// TIA Portal project "LogicRoof" (V17)

(* hardware
DEVICE "S7-1500/ET200MP station_1"  S7-1500 station
   slot 0: "Rail_0"  Rack  6ES7 590-1***0-0AA0
   slot 1: "MAIN_PLC"  CPU 1517F-3 PN/DP  6ES7 517-3FP00-0AB0  V2.9
      slot 3: "CPU display_1"  6ES7591-1BA00-0AA0
      slot 32768: "PROFINET interface_1"  X1
         slot 32769: "Port_1"  X1 P1
         slot 32770: "Port_2"  X1 P2
      slot 33024: "PROFINET interface_2"  X2
         slot 33025: "Port_1"  X2 P1
      slot 33280: "DP interface_1"  X3
      slot 34817: "Virtual CP interface port_1"  Virtual CP interface port  Virtual CP interface port
   slot 2: "CP 1543-1_1"  CP 1543-1  6GK7 543-1AX00-0XE0  V3.0
DEVICE "Lift1_PLC"  GSD.Device.PN
   slot 0: "Rack"  Rack  V1.0
   slot 1: "Lift1_PLC"  PLC-Lift1  6ES7 288-1ST60-0AA1  V02.07.00
      slot 0: "PLC-Lift1 Virtual submodule"  PLC-Lift1 Virtual submodule
      slot 1: "传送区01"  传送区01
      slot 2: "传送区02"  传送区02
      slot 3: "Interface"  Interface
         slot 1: "Port 1"  Port 1
DEVICE "Stacker_PLC"  GSD.Device.PN
   slot 0: "Rack"  Rack  V1.0
   slot 1: "Stacker_PLC"  PLC-Stacker  6ES7 288-1ST60-0AA0  V02.05.00
      slot 0: "PLC-Stacker Virtual submodule"  PLC-Stacker Virtual submodule
      slot 1: "传送区01"  传送区01
      slot 2: "传送区02"  传送区02
      slot 3: "Interface"  Interface
         slot 1: "Port 1"  Port 1
DEVICE "MDB_IO"  GSD.Device.PN
   slot 0: "Rack"  Rack  V1.0
   slot 0: "mdb-io"  CN-8032  CN-8032  V1.00
      slot 0: "CN-8032"  CN-8032
      slot 1: "PN-IO"  PN-IO
         slot 1: "Port 1"  Port 1
         slot 2: "Port 2"  Port 2
   slot 1: "DI1"  CT-121F (16DI 24Vdc) Sink Input  CT-121F  V1.00
      slot 0: "16DI Input Status"  16DI Input Status
   slot 1: "16DI Counter Submodule"  16DI Counter Submodule
   slot 1: "16DI Counter Submodule"  16DI Counter Submodule
   slot 2: "DI2"  CT-121F (16DI 24Vdc) Sink Input  CT-121F  V1.00
      slot 0: "16DI Input Status"  16DI Input Status
   slot 3: "DI3"  CT-121F (16DI 24Vdc) Sink Input  CT-121F  V1.00
      slot 0: "16DI Input Status"  16DI Input Status
   slot 4: "DO1"  CT-222F (16DO 24Vdc) Source Output TTL  CT-222F  V1.00
      slot 0: "16DO Output Status"  16DO Output Status
   slot 5: "DO2"  CT-222F (16DO 24Vdc) Source Output TTL  CT-222F  V1.00
      slot 0: "16DO Output Status"  16DO Output Status
DEVICE "SDB_IO"  GSD.Device.PN
   slot 0: "Rack"  Rack  V1.0
   slot 0: "SDB-IO"  CN-8032  CN-8032  V1.00
      slot 0: "CN-8032"  CN-8032
      slot 1: "PN-IO"  PN-IO
         slot 1: "Port 1"  Port 1
         slot 2: "Port 2"  Port 2
   slot 1: "DI1"  CT-121F (16DI 24Vdc) Sink Input  CT-121F  V1.00
      slot 0: "16DI Input Status"  16DI Input Status
   slot 1: "16DI Counter Submodule"  16DI Counter Submodule
   slot 1: "16DI Counter Submodule"  16DI Counter Submodule
   slot 2: "DI2"  CT-121F (16DI 24Vdc) Sink Input  CT-121F  V1.00
      slot 0: "16DI Input Status"  16DI Input Status
   slot 4: "DO1"  CT-222F (16DO 24Vdc) Source Output TTL  CT-222F  V1.00
      slot 0: "16DO Output Status"  16DO Output Status
DEVICE "PU_IO"  GSD.Device.PN
   slot 0: "Rack"  Rack  V1.0
   slot 0: "PU-IO"  CN-8032  CN-8032  V1.00
      slot 0: "CN-8032"  CN-8032
      slot 1: "PN-IO"  PN-IO
         slot 1: "Port 1"  Port 1
         slot 2: "Port 2"  Port 2
   slot 1: "DI1"  CT-121F (16DI 24Vdc) Sink Input  CT-121F  V1.00
      slot 0: "16DI Input Status"  16DI Input Status
   slot 1: "16DI Counter Submodule"  16DI Counter Submodule
   slot 1: "16DI Counter Submodule"  16DI Counter Submodule
   slot 4: "DO1"  CT-222F (16DO 24Vdc) Source Output TTL  CT-222F  V1.00
      slot 0: "16DO Output Status"  16DO Output Status
DEVICE "Lift2_PLC"  GSD.Device.PN
   slot 0: "Rack"  Rack  V1.0
   slot 1: "Lift2_PLC"  PLC-Lift1  6ES7 288-1ST60-0AA1  V02.07.00
      slot 0: "PLC-Lift1 Virtual submodule"  PLC-Lift1 Virtual submodule
      slot 1: "传送区01"  传送区01
      slot 2: "传送区02"  传送区02
      slot 3: "Interface"  Interface
         slot 1: "Port 1"  Port 1
DEVICE "GSD device_1"  GSD.Device.PN
   slot 0: "Rack"  Rack  V1.0
   slot 0: "C8-U1"  ConveyLinx in PLC mode  ERSC  V5.07.00
      slot 0: "ConveyLinx in PLC mode"  ConveyLinx in PLC mode
      slot 1: "Interface"  Interface
         slot 1: "Port 1"  Port 1
         slot 2: "Port 2"  Port 2
      slot 1: "Inputs"  virtual input module 64 byte  NO_ORDER_CODE  1.0
         slot 0: "virtual input module 64 byte"  virtual input module 64 byte
      slot 2: "Outputs"  virtual output module 64 byte  NO_ORDER_CODE  1.0
         slot 0: "virtual output module 64 byte"  virtual output module 64 byte
DEVICE "C1_M1_1"  GSD.Device.PN
   slot 0: "Rack"  Rack  V1.0
   slot 0: "C2-M1"  AD1000PN  AD1000PN
      slot 0: "AD1000PN"  AD1000PN
      slot 1: "Interface"  Interface
         slot 1: "Port 1"  Port 1
         slot 2: "Port 2"  Port 2
   slot 1: "Data"  Standard telegram 3, PZD-6/6
      slot 0: "Standard telegram 3, PZD-6/6"  Standard telegram 3, PZD-6/6
DEVICE "C1_M1_2"  GSD.Device.PN
   slot 0: "Rack"  Rack  V1.0
   slot 0: "C1-M1"  AD1000PN  AD1000PN
      slot 0: "AD1000PN"  AD1000PN
      slot 1: "Interface"  Interface
         slot 1: "Port 1"  Port 1
         slot 2: "Port 2"  Port 2
   slot 1: "Data"  Standard telegram 3, PZD-6/6
      slot 0: "Standard telegram 3, PZD-6/6"  Standard telegram 3, PZD-6/6
*)

// ===== PLC "MAIN_PLC"  CPU 1517F-3 PN/DP =====

VAR_GLOBAL   // PLC tag table "SDB_IO"
   "bSDB_KM1_St" AT %I218.0 : Bool;   // Статус главного контактора
   "bSDB_QF1_St" AT %I218.1 : Bool;   // Статус автоматического выкл. QF1
   "bSDB_QF2_St" AT %I218.2 : Bool;   // Статус автоматического выкл. QF2
   "bSDB_QF3_St" AT %I218.3 : Bool;   // Статус автоматического выкл. QF3
   "bSDB_QF4_St" AT %I218.4 : Bool;   // Статус автоматического выкл. QF4
   "bSDB_QF5_St" AT %I218.5 : Bool;   // Статус автоматического выкл. QF5
   "bSDB_QF6_St" AT %I218.6 : Bool;   // Статус автоматического выкл. QF6
   "bFS_SDB_KSF1_St" AT %I218.7 : Bool;   // Статус реле безопасности KSF1
   "bFS_SDB_SB2_St" AT %I219.0 : Bool;   // Кнопка аварийного останова
   "bFS_SDB_SBR1_St" AT %I219.1 : Bool;   // Кнопка сброса аварии
   "bFS_SR3_St" AT %I219.2 : Bool;   // Трос безопасности SR3
   "bFS_SR3_1_St" AT %I219.3 : Bool;   // Трос безопасности SR3.1
   "bFS_SR3_2_St" AT %I219.4 : Bool;   // Трос безопасности SR3.2
   "bFS_SR3_3_St" AT %I219.5 : Bool;   // Трос безопасности SR3.3
   "bSens_5_D4" AT %I219.6 : Bool;   // Датчик -5-D4
   "bSens_5_D5" AT %I219.7 : Bool;   // Датчик -5-D5
   "bSens_6_D4" AT %I284.0 : Bool;   // Датчик -6-D4
   "bSens_6_D5" AT %I284.1 : Bool;   // Датчик -6-D5
   "bSens_7_D4" AT %I284.2 : Bool;   // Датчик -7-D4
   "bSens_7_D5" AT %I284.3 : Bool;   // Датчик -7-D5
   "bSens_8_D3" AT %I284.4 : Bool;   // Датчик -8-D3
   "bFS_SB4_St" AT %I284.5 : Bool;   // Кнопка аварийного останова SB4
   "bFS_SB5_St" AT %I284.6 : Bool;   // Кнопка аварийного останова SB5
   "bFS_SB6_St" AT %I284.7 : Bool;   // Кнопка аварийного останова SB6
   "bFS_SB7_St" AT %I285.0 : Bool;   // Кнопка аварийного останова SB7
   "bSDB_DI2_9" AT %I285.1 : Bool;   // Резерв
   "bSDB_DI2_10" AT %I285.2 : Bool;   // Резерв
   "bSDB_DI2_11" AT %I285.3 : Bool;   // Резерв
   "bSDB_DI2_12" AT %I285.4 : Bool;   // Резерв
   "bSDB_DI2_13" AT %I285.5 : Bool;   // Резерв
   "bSDB_DI2_14" AT %I285.6 : Bool;   // Резерв
   "bSDB_DI2_15" AT %I285.7 : Bool;   // Резерв
   "bSDB_KM1_Ctrl" AT %Q90.0 : Bool;   // Вкл. главного контактора
   "bFS_SDB_KSF1_Reset" AT %Q90.1 : Bool;   // Сброс реле безопасности (старт)
   "bFS_SDB_SafetyMuting" AT %Q90.2 : Bool;   // Safety muting
   "bFS_Lift1Safety_Reset" AT %Q90.3 : Bool;   // Сброс реле безопасности (старт) Лифта 1
   "bSDB_DO1_4" AT %Q90.4 : Bool;   // Резерв
   "bSDB_DO1_5" AT %Q90.5 : Bool;   // Резерв
   "bSDB_DO1_6" AT %Q90.6 : Bool;   // Резерв
   "bSDB_DO1_7" AT %Q90.7 : Bool;   // Резерв
   "bSDB_GeneralAlarm_Ind" AT %Q91.0 : Bool;   // Общая авария
   "bFS_SDB_SafetyAlarm_Ind" AT %Q91.1 : Bool;   // Авария системы безопасности
   "bFS_SDB_SBR1_HL" AT %Q91.2 : Bool;   // Подсветка кнопки СБРОС
   "bSDB_Light_Red" AT %Q91.3 : Bool;   // Свет. колонна, Красный
   "bSDB_Light_Yellow" AT %Q91.4 : Bool;   // Свет. колонна, Желтый
   "bSDB_Light_Green" AT %Q91.5 : Bool;   // Свет. колонна, Зеленый
   "bSDB_Light_Blue" AT %Q91.6 : Bool;   // Свет. колонна, Синий
   "bSDB_Light_Siren" AT %Q91.7 : Bool;   // Свет. колонна, Сирена
END_VAR

VAR_GLOBAL   // PLC tag table "MDB_IO"
   "bStation1_Pwr_St" AT %I64.0 : Bool;   // Цепь питания станции вызревания 1
   "bStation2_Pwr_St" AT %I64.1 : Bool;   // Цепь питания станции вызревания 2
   "bStation3_Pwr_St" AT %I64.2 : Bool;   // Цепь питания станции вызревания 3
   "bStation4_Pwr_St" AT %I64.3 : Bool;   // Цепь питания станции вызревания 4
   "bStation5_Pwr_St" AT %I64.4 : Bool;   // Цепь питания станции вызревания 5
   "bStation6_Pwr_St" AT %I64.5 : Bool;   // Цепь питания станции вызревания 6
   "bStation7_Pwr_St" AT %I64.6 : Bool;   // Цепь питания станции вызревания 7
   "bStation8_Pwr_St" AT %I64.7 : Bool;   // Цепь питания станции вызревания 8
   "bStation9_Pwr_St" AT %I65.0 : Bool;   // Цепь питания станции вызревания 9
   "bStation10_Pwr_St" AT %I65.1 : Bool;   // Цепь питания станции вызревания 10
   "bStation11_Pwr_St" AT %I65.2 : Bool;   // Цепь питания станции вызревания 11
   "bStation12_Pwr_St" AT %I65.3 : Bool;   // Цепь питания станции вызревания 12
   "bStation13_Pwr_St" AT %I65.4 : Bool;   // Цепь питания станции вызревания 13
   "bStation14_Pwr_St" AT %I65.5 : Bool;   // Цепь питания станции вызревания 14
   "bConv35_36_Pwr_St" AT %I65.6 : Bool;   // Автомат QF15 питания шкафа SDB включен
   "bMDB_QF16_St" AT %I65.7 : Bool;   // Автомат QF16 питания паллетайзера включен
   "bMDB_QF17_St" AT %I150.0 : Bool;   // Автомат QF17 питания лифта 2
   "bMDB_QF18_St" AT %I150.1 : Bool;   // Автомат QF18 питания секций 35, 36
   "bMDB_K1_St" AT %I150.2 : Bool;   // Реле контроля фаз K1
   "bFS_MDB_KSF1_St" AT %I150.3 : Bool;   // Статус реле безопасности KSF1
   "bFS_MDB_KSF2_St" AT %I150.4 : Bool;   // Статус реле безопасности KSF2
   "bFS_MDB_KSF3_St" AT %I150.5 : Bool;   // Статус реле безопасности KSF3
   "bFS_MDB_SB1_St" AT %I150.6 : Bool;   // Кнопка аварийного останова SB1
   "bFS_MDB_SBR1_St" AT %I150.7 : Bool;   // Кнопка сброса аварии SBR1
   "bFS_SR1_St" AT %I151.0 : Bool;   // Трос безопасности SR1
   "bFS_SR1_1_St" AT %I151.1 : Bool;   // Трос безопасности SR1.1
   "bFS_SR1_2_St" AT %I151.2 : Bool;   // Трос безопасности SR1.2
   "bFS_SR1_3_St" AT %I151.3 : Bool;   // Трос безопасности SR1.3
   "bFS_SR2_St" AT %I151.4 : Bool;   // Трос безопасности SR2
   "bFS_SR2_1_St" AT %I151.5 : Bool;   // Трос безопасности SR2.1
   "bFS_SR2_2_St" AT %I151.6 : Bool;   // Трос безопасности SR2.2
   "bFS_SR2_3_St" AT %I151.7 : Bool;   // Трос безопасности SR2.3
   "bSens_37_D1" AT %I216.0 : Bool;   // Датчик 37-D1
   "bSens_37_D2" AT %I216.1 : Bool;   // Датчик 37-D2
   "bSens_37_D4" AT %I216.2 : Bool;   // Датчик 37-D4
   "bSens_37_D5" AT %I216.3 : Bool;   // Датчик 37-D5
   "bSens_37_D3" AT %I216.4 : Bool;   // Датчик 37-D3
   "bMDB_DI3_5" AT %I216.5 : Bool;   // Резерв 1
   "bMDB_DI3_6" AT %I216.6 : Bool;   // Резерв 2
   "bMDB_DI3_7" AT %I216.7 : Bool;   // Резерв 3
   "bMDB_DI3_8" AT %I217.0 : Bool;   // Резерв 4
   "bMDB_DI3_9" AT %I217.1 : Bool;   // Резерв 5
   "bMDB_DI3_10" AT %I217.2 : Bool;   // Резерв 6
   "bMDB_DI3_11" AT %I217.3 : Bool;   // Резерв 7
   "bMDB_DI3_12" AT %I217.4 : Bool;   // Резерв 8
   "bMDB_DI3_13" AT %I217.5 : Bool;   // Резерв 9
   "bMDB_DI3_14" AT %I217.6 : Bool;   // Резерв 10
   "bMDB_DI3_15" AT %I217.7 : Bool;   // Резерв 11
   "bStation1_Pwr_Ctrl" AT %Q82.0 : Bool;   // Вкл. cтанции вызревания 1
   "bStation2_Pwr_Ctrl" AT %Q82.1 : Bool;   // Вкл. cтанции вызревания 2
   "bStation3_Pwr_Ctrl" AT %Q82.2 : Bool;   // Вкл. cтанции вызревания 3
   "bStation4_Pwr_Ctrl" AT %Q82.3 : Bool;   // Вкл. cтанции вызревания 4
   "bStation5_Pwr_Ctrl" AT %Q82.4 : Bool;   // Вкл. cтанции вызревания 5
   "bStation6_Pwr_Ctrl" AT %Q82.5 : Bool;   // Вкл. cтанции вызревания 6
   "bStation7_Pwr_Ctrl" AT %Q82.6 : Bool;   // Вкл. cтанции вызревания 7
   "bStation8_Pwr_Ctrl" AT %Q82.7 : Bool;   // Вкл. cтанции вызревания 8
   "bStation9_Pwr_Ctrl" AT %Q83.0 : Bool;   // Вкл. cтанции вызревания 9
   "bStation10_Pwr_Ctrl" AT %Q83.1 : Bool;   // Вкл. cтанции вызревания 10
   "bStation11_Pwr_Ctrl" AT %Q83.2 : Bool;   // Вкл. cтанции вызревания 11
   "bStation12_Pwr_Ctrl" AT %Q83.3 : Bool;   // Вкл. cтанции вызревания 12
   "bStation13_Pwr_Ctrl" AT %Q83.4 : Bool;   // Вкл. cтанции вызревания 13
   "bStation14_Pwr_Ctrl" AT %Q83.5 : Bool;   // Вкл. cтанции вызревания 14
   "bConv35_36_Pwr_Ctrl" AT %Q83.6 : Bool;   // Вкл. трансфера и ролик.конвейера
   "bMDB_DO1_15" AT %Q83.7 : Bool;   // Резерв
   "bMDB_GeneralAlarm_Ind" AT %Q84.0 : Bool;   // Общая авария
   "bFS_MDB_SafetyAlarm_Ind" AT %Q84.1 : Bool;   // Авария системы безопасности
   "bFS_MDB_SBR1_HL" AT %Q84.2 : Bool;   // Подсветка кнопки "Сброс"
   "bMDB_Light_Red" AT %Q84.3 : Bool;   // Свет. колонна, Красный
   "bMDB_Light_Yellow" AT %Q84.4 : Bool;   // Свет. колонна, Желтый
   "bMDB_Light_Green" AT %Q84.5 : Bool;   // Свет. колонна, Зеленый
   "bMDB_Light_Blue" AT %Q84.6 : Bool;   // Свет. колонна, Синий
   "bMDB_Light_Siren" AT %Q84.7 : Bool;   // Свет. колонна, Сирена
   "bFS_MDB_KSF1_2_Reset" AT %Q85.0 : Bool;   // Сброс реле безопасности (старт) KSF1 и KSF2
   "bFS_MDB_KSF3_Reset" AT %Q85.1 : Bool;   // Сброс реле безопасности (старт) KSF3
   "bFS_MDB_SafetyMuting" AT %Q85.2 : Bool;   // Safety muting
   "bFS_Lift2Safety_Reset" AT %Q85.3 : Bool;   // Сброс реле безопасности (старт) Лифта 2
   "bFS_StackerSafety_Reset" AT %Q85.4 : Bool;   // Сброс реле безопасности (старт) трехкоординатного стекера
   "bMDB_DO2_13" AT %Q85.5 : Bool;   // Резерв
   "bMDB_DO2_14" AT %Q85.6 : Bool;   // Резерв
   "bMDB_DO2_15" AT %Q85.7 : Bool;   // Резерв
END_VAR

VAR_GLOBAL   // PLC tag table "PU_IO"
   "bFS_PU_SB3_St" AT %I4.0 : Bool;   // Кнопка аварийного останова
   "bFS_PU_SBR1_St" AT %I4.1 : Bool;   // Кнопка сброса аварии
   "bSens_3_S1" AT %I4.2 : Bool;   // Датчик -3-S1
   "bSens_3_S2" AT %I4.3 : Bool;   // Датчик -3-S2
   "bPU_DI1_4" AT %I4.4 : Bool;   // Резерв
   "bPU_DI1_5" AT %I4.5 : Bool;   // Резерв
   "bPU_DI1_6" AT %I4.6 : Bool;   // Резерв
   "bPU_DI1_7" AT %I4.7 : Bool;   // Резерв
   "bPU_DI1_8" AT %I5.0 : Bool;   // Резерв
   "bPU_DI1_9" AT %I5.1 : Bool;   // Резерв
   "bPU_DI1_10" AT %I5.2 : Bool;   // Резерв
   "bPU_DI1_11" AT %I5.3 : Bool;   // Резерв
   "bPU_DI1_12" AT %I5.4 : Bool;   // Резерв
   "bPU_DI1_13" AT %I5.5 : Bool;   // Резерв
   "bPU_DI1_14" AT %I5.6 : Bool;   // Резерв
   "bPU_DI1_15" AT %I5.7 : Bool;   // Резерв
   "bPU_GeneralAlarm_Ind" AT %I6.0 : Bool;   // Общая авария
   "bFS_PU_SafetyAlarm_Ind" AT %I6.1 : Bool;   // Авария системы безопасности
   "bFS_PU_SBR1_HL" AT %I6.2 : Bool;   // Подсветка кнопки СБРОС
   "bPU_DO1_3" AT %I6.3 : Bool;   // Резерв
   "bPU_DO1_4" AT %I6.4 : Bool;   // Резерв
   "bPU_DO1_5" AT %I6.5 : Bool;   // Резерв
   "bPU_DO1_6" AT %I6.6 : Bool;   // Резерв
   "bPU_DO1_7" AT %I6.7 : Bool;   // Резерв
   "bPU_DO1_8" AT %I7.0 : Bool;   // Резерв
   "bPU_DO1_9" AT %I7.1 : Bool;   // Резерв
   "bPU_DO1_10" AT %I7.2 : Bool;   // Резерв
   "bPU_DO1_11" AT %I7.3 : Bool;   // Резерв
   "bPU_DO1_12" AT %I7.4 : Bool;   // Резерв
   "bPU_DO1_13" AT %I7.5 : Bool;   // Резерв
   "bPU_DO1_14" AT %I7.6 : Bool;   // Резерв
   "bPU_DO1_15" AT %I7.7 : Bool;   // Резерв
END_VAR

VAR_GLOBAL   // PLC tag table "Drives"
   "Drive01_M1" AT %I0.0 : "stDriveType";
END_VAR

VAR_GLOBAL   // PLC tag table "Global"
   "bResetAlarm" AT %M0.0 : Bool;
   "bRd" AT %M0.1 : Bool;
   "vrRec" AT %MW12 : Word;
   "Tag_1" AT %MW14 : Int;
   "Tag_2" AT %MW16 : Int;
END_VAR

TYPE "stOutbound"
   STRUCT
      bMove : Bool;
      bAllowMove : Bool;
      byConvStatus : Byte;
      bReverse : Bool;
   END_STRUCT;
END_TYPE

TYPE "stDriveType"
   STRUCT
      bDrive : Bool;   // Drive forward output
      bDriveRev : Bool;   // Drive reverse output
      bLowSpeed : Bool;   // Low speed select
      bAlarm : Bool;   // General alarm
      bButtDrive : Bool;   // Manual drive button
      bButtDriveRev : Bool;   // Manual reverse drive button
      bLock : Bool;   // Locking motor
      bSafety : Bool;
      bSwitch : Bool;
      bReadyToRun : Bool;
      bNotReady : Bool;
   END_STRUCT;
END_TYPE

TYPE "stModeType"
   STRUCT
      bAutomat : Bool;   // Auto mode
      bStartAutomat : Bool;   // Auto starting mode
      bStop : Bool;   // Stop mode
      bManual : Bool;   // Manual mode
      bReset : Bool;   // Reset mode
      bResetAlarm : Bool;   // Reset alarms
      bAlarm : Bool;   // Alarm mode
      bReadyToReset : Bool;   // Ready to reset mode
   END_STRUCT;
END_TYPE

TYPE "stDriveIOType"
   STRUCT
      uiIn1 : Int;
      uiIn2 : Int;
      uiIn3 : Int;
      uiIn4 : Int;
      uiIn5 : Int;
      uiIn6 : Int;
      uiOut1 : Int;
      uiOut2 : Int;
      uiOut3 : Int;
      uiOut4 : Int;
      uiOut5 : Int;
      uiOut6 : Int;
   END_STRUCT;
END_TYPE

TYPE "stOutboundRev"
   STRUCT
      bMove : Bool;
      bAllowMove : Bool;
      bMoveRev : Bool;
      bAllowMoveRev : Bool;
      byConvStatus : Byte;
      bReverse : Bool;
   END_STRUCT;
END_TYPE

// folder: FB_DB

DATA_BLOCK "FB_Light_DB"   // DB19
{ S7_Optimized_Access := 'TRUE' }
VERSION : 0.1
// stored: InstanceOfName FB_Light
"FB_Light"
BEGIN
END_DATA_BLOCK

DATA_BLOCK "FB_Mode_DB"   // DB20
{ S7_Optimized_Access := 'TRUE' }
VERSION : 0.1
// stored: InstanceOfName FB_Mode
"FB_Mode"
BEGIN
END_DATA_BLOCK

DATA_BLOCK "FB_SystemTime_DB"   // DB24
{ S7_Optimized_Access := 'TRUE' }
VERSION : 0.1
// stored: InstanceOfName FB_SystemTime
"FB_SystemTime"
BEGIN
END_DATA_BLOCK

// folder: FB_DB/Conv

DATA_BLOCK "fbConv_001"   // DB21
{ S7_Optimized_Access := 'TRUE' }
VERSION : 0.1
// stored: InstanceOfName FB_DirectSection
"FB_DirectSection"
BEGIN
END_DATA_BLOCK

DATA_BLOCK "fbConv_002"   // DB22
{ S7_Optimized_Access := 'TRUE' }
VERSION : 0.1
// stored: InstanceOfName FB_DirectSection
"FB_DirectSection"
BEGIN
END_DATA_BLOCK

DATA_BLOCK "fbConv_010"   // DB23
{ S7_Optimized_Access := 'TRUE' }
VERSION : 0.1
// stored: InstanceOfName FB_DirectSection
"FB_DirectSection"
BEGIN
END_DATA_BLOCK

DATA_BLOCK "fbConv_004"   // DB25
{ S7_Optimized_Access := 'TRUE' }
VERSION : 0.1
// stored: InstanceOfName FB_DirectSectionRev
"FB_DirectSectionRev"
BEGIN
END_DATA_BLOCK

DATA_BLOCK "fbConv_003"   // DB26
{ S7_Optimized_Access := 'TRUE' }
VERSION : 0.1
// stored: InstanceOfName FB_RotarySection
"FB_RotarySection"
BEGIN
END_DATA_BLOCK

DATA_BLOCK "fbConv_009"   // DB27
{ S7_Optimized_Access := 'TRUE' }
VERSION : 0.1
// stored: InstanceOfName FB_DirectSection
"FB_DirectSection"
BEGIN
END_DATA_BLOCK

// folder: Safety

DATA_BLOCK "FB_SafetyGroup_DB"   // DB4
{ S7_Optimized_Access := 'TRUE' }
VERSION : 0.1
// stored: InstanceOfName FB_SafetyGroup
"FB_SafetyGroup"
BEGIN
END_DATA_BLOCK

// folder: Safety/PWR

DATA_BLOCK "FB_Station1Pwr_DB"   // DB1
{ S7_Optimized_Access := 'TRUE' }
VERSION : 0.1
// stored: InstanceOfName FB_PowerGroup
"FB_PowerGroup"
BEGIN
END_DATA_BLOCK

DATA_BLOCK "FB_Station2Pwr_DB"   // DB2
{ S7_Optimized_Access := 'TRUE' }
VERSION : 0.1
// stored: InstanceOfName FB_PowerGroup
"FB_PowerGroup"
BEGIN
END_DATA_BLOCK

DATA_BLOCK "FB_Station7Pwr_DB"   // DB3
{ S7_Optimized_Access := 'TRUE' }
VERSION : 0.1
// stored: InstanceOfName FB_PowerGroup
"FB_PowerGroup"
BEGIN
END_DATA_BLOCK

DATA_BLOCK "FB_Station8Pwr_DB"   // DB5
{ S7_Optimized_Access := 'TRUE' }
VERSION : 0.1
// stored: InstanceOfName FB_PowerGroup
"FB_PowerGroup"
BEGIN
END_DATA_BLOCK

DATA_BLOCK "FB_Station9Pwr_DB"   // DB6
{ S7_Optimized_Access := 'TRUE' }
VERSION : 0.1
// stored: InstanceOfName FB_PowerGroup
"FB_PowerGroup"
BEGIN
END_DATA_BLOCK

DATA_BLOCK "FB_Station10Pwr_DB"   // DB7
{ S7_Optimized_Access := 'TRUE' }
VERSION : 0.1
// stored: InstanceOfName FB_PowerGroup
"FB_PowerGroup"
BEGIN
END_DATA_BLOCK

DATA_BLOCK "FB_Station11Pwr_DB"   // DB8
{ S7_Optimized_Access := 'TRUE' }
VERSION : 0.1
// stored: InstanceOfName FB_PowerGroup
"FB_PowerGroup"
BEGIN
END_DATA_BLOCK

DATA_BLOCK "FB_Station12Pwr_DB"   // DB9
{ S7_Optimized_Access := 'TRUE' }
VERSION : 0.1
// stored: InstanceOfName FB_PowerGroup
"FB_PowerGroup"
BEGIN
END_DATA_BLOCK

DATA_BLOCK "FB_Station13Pwr_DB"   // DB10
{ S7_Optimized_Access := 'TRUE' }
VERSION : 0.1
// stored: InstanceOfName FB_PowerGroup
"FB_PowerGroup"
BEGIN
END_DATA_BLOCK

DATA_BLOCK "FB_Conv35_36Pwr_DB"   // DB11
{ S7_Optimized_Access := 'TRUE' }
VERSION : 0.1
// stored: InstanceOfName FB_PowerGroup
"FB_PowerGroup"
BEGIN
END_DATA_BLOCK

DATA_BLOCK "FB_Station5Pwr_DB"   // DB12
{ S7_Optimized_Access := 'TRUE' }
VERSION : 0.1
// stored: InstanceOfName FB_PowerGroup
"FB_PowerGroup"
BEGIN
END_DATA_BLOCK

DATA_BLOCK "FB_SDB_KM1Pwr_DB"   // DB13
{ S7_Optimized_Access := 'TRUE' }
VERSION : 0.1
// stored: InstanceOfName FB_PowerGroup
"FB_PowerGroup"
BEGIN
END_DATA_BLOCK

DATA_BLOCK "FB_Station3Pwr_DB"   // DB14
{ S7_Optimized_Access := 'TRUE' }
VERSION : 0.1
// stored: InstanceOfName FB_PowerGroup
"FB_PowerGroup"
BEGIN
END_DATA_BLOCK

DATA_BLOCK "FB_Station14Pwr_DB"   // DB15
{ S7_Optimized_Access := 'TRUE' }
VERSION : 0.1
// stored: InstanceOfName FB_PowerGroup
"FB_PowerGroup"
BEGIN
END_DATA_BLOCK

DATA_BLOCK "FB_Station4Pwr_DB"   // DB16
{ S7_Optimized_Access := 'TRUE' }
VERSION : 0.1
// stored: InstanceOfName FB_PowerGroup
"FB_PowerGroup"
BEGIN
END_DATA_BLOCK

DATA_BLOCK "FB_Station6Pwr_DB"   // DB17
{ S7_Optimized_Access := 'TRUE' }
VERSION : 0.1
// stored: InstanceOfName FB_PowerGroup
"FB_PowerGroup"
BEGIN
END_DATA_BLOCK

// folder: System blocks/Program resources

DATA_BLOCK "FB_StartTimer_DB"   // DB18
{ S7_Optimized_Access := 'TRUE' }
AUTHOR : Simatic
FAMILY : IEC
NAME : IEC_TMR
VERSION : 1.0
// stored: InstanceOfName IEC_TIMER
"IEC_TIMER"
BEGIN
END_DATA_BLOCK

// folder: (top level)

FUNCTION_BLOCK "FB_DirectSection_OLD"   // FB13, SCL
{ S7_Optimized_Access := 'FALSE' }
VERSION : 0.1
   VAR_INPUT
      bStartAutomat : Bool;
      bFinalConv : Bool := true;
      bFinalConvReverse : Bool := true;
      bAutomat : Bool;
      bEnable1 : Bool;
      tStartTimer : Time := T#20s;
      bEnable2 : Bool;
      bEnable3 : Bool;
      bEnable4 : Bool;
      ConvStatusPrev : Byte;
      ConvStatusNext : Byte;
      bManual : Bool;
      bDriveAuto : Bool;
      bDriveAutoReverse : Bool;
      bButtManu : Bool;
      bButtManuReverse : Bool;
      bButtMove : Bool;
      bButtMoveReverse : Bool;
      bSens : Bool;
      bSens2 : Bool;
      bSens3 : Bool := true;
      bSensFork : Bool;
      tBusy : Time := T#0.01s;
      tFree : Time := T#3s;
      tLongMove : Time := T#40s;
      bReset : Bool;
      bStop : Bool;
      bReverse : Bool;
      bCurtaineUp : Bool := true;
   END_VAR
   VAR_OUTPUT
      bDrive : Bool;
      bDriveReverse : Bool;
      ConvStatus : Byte;
      bDrivePrev : Bool;
      bLongMoveReverse : Bool;
      bLongMove : Bool;
      bDriveNext : Bool;
      bMovePerm : Bool;
      bMovePermRev : Bool;
   END_VAR
   VAR_IN_OUT
      bMove : Bool;
      bMoveReverse : Bool;
   END_VAR
   VAR
      bDriveManu : Bool;
      bResManu : Bool;
      bDriveManuReverse : Bool;
      bDriveConv : Bool;
      bOnMove : Bool;
      bOffMove : Bool;
      bDriveConvReverse : Bool;
      bOnMoveReverse : Bool;
      bOffMoveReverse : Bool;
      bStartConv : Bool;
      bStartConvReverse : Bool;
      fbBusy1 : "FB_Busy1_LAD";
      fbBusy2 : "FB_Busy1_LAD";
      fbBusy3 : "FB_Busy1_LAD";
      fbBusyFork : "FB_Busy2_LAD";
      fbButt : "FB_Button";
      fbButtReverse : "FB_Button";
      fbLongMove : TON_TIME;
      fbLongMoveReverse : TON_TIME;
      fbButtMove : "FB_r_trig";
      fbButtMoveReverse : "FB_r_trig";
      fbStartAutomat : "FB_r_trig";
      fbConvBusy1Puls : "FB_r_trig";
      fbConvBusy2Puls : "FB_r_trig";
      fbStartTimer : TON_TIME;
      fbStartTimerReverse : TON_TIME;
   END_VAR
BEGIN
   #fbBusy1(bSens:= #bSens,  tFree:=  #tFree ,   tBusy:= #tBusy , Reset := #bReset );
   #fbBusy2(bSens:= #bSens2,  tFree:=   #tFree ,   tBusy:=  #tBusy , Reset := #bReset);
   #fbBusy3( bSens:= #bSens3,  tFree:=   #tFree ,   tBusy:=  #tBusy , Reset := #bReset);
   #fbBusyFork(bSens:= #bSensFork,  tFree:=   T#5s ,   tBusy:= T#0s , Reset := #bReset);

   IF NOT #fbBusy1.ConvBusy AND NOT #fbBusy2.ConvBusy AND #bSens3 THEN
       #ConvStatus := 0;
   ELSIF #fbBusy1.ConvBusy AND NOT #fbBusy2.ConvBusy THEN
       #ConvStatus := 1;
   ELSIF NOT #fbBusy1.ConvBusy AND #fbBusy2.ConvBusy THEN
       #ConvStatus := 2;
   ELSIF #fbBusy1.ConvBusy AND #fbBusy2.ConvBusy THEN
       #ConvStatus := 3;
   END_IF;

   #bDrive := NOT #bStop AND (#bDriveAuto OR #bDriveConv OR #bDriveManu OR #bStartConv);
   #bDriveReverse := NOT #bStop AND (#bDriveAutoReverse OR #bDriveConvReverse OR #bDriveManuReverse OR #bStartConvReverse);

   #bResManu := #bReset OR NOT #bManual;
   #fbButt(bBut:=#bButtManu AND #bManual AND NOT #bDriveManuReverse,
           bRS:= #bResManu,
           bOutB=>#bDriveManu);
   #fbButtReverse(bBut:=#bButtManuReverse AND #bManual  AND NOT #bDriveManu,
                  bRS:=#bResManu,
                  bOutB=>#bDriveManuReverse);
   (*перемещение*)
   (* условия включения перемещения*)
   #bMovePerm := #bAutomat AND #bEnable1 AND #bEnable2 AND (#ConvStatusPrev = 2 OR #ConvStatusPrev = 3) AND #ConvStatus = 0 AND NOT #fbBusyFork.ConvBusy AND NOT #bReverse;
   IF #bMovePerm AND #bCurtaineUp
   THEN
       #bMove := TRUE;
   END_IF;
   (* условия включения обратного перемещения *)
   #bMovePermRev := #bAutomat AND #bEnable3 AND #bEnable4 AND (#ConvStatusNext = 1 OR #ConvStatusNext = 3) AND #ConvStatus = 0 AND NOT #fbBusyFork.ConvBusy AND #bReverse;
   IF #bMovePermRev AND #bCurtaineUp
   THEN
       #bMoveReverse := TRUE;
   END_IF;
   (* включение двигателей *)
   #bDriveConv := NOT #bStop AND #bMove AND NOT (#ConvStatus = 2 OR #ConvStatus = 3);
   #bDrivePrev := NOT #bStop AND #bMove AND NOT (#ConvStatus = 2 OR #ConvStatus = 3) AND NOT (#ConvStatusPrev = 0);
   (* включение двигателей при реверсе*)
   #bDriveConvReverse := NOT #bStop AND #bMoveReverse AND NOT (#ConvStatus = 1 OR #ConvStatus = 3);
   #bDriveNext := NOT #bStop AND #bMoveReverse AND NOT (#ConvStatus = 1 OR #ConvStatus = 3) AND NOT (#ConvStatusNext = 0);
   (* выключение перемещения*)
   IF #bMove AND #ConvStatusPrev = 0 AND (#ConvStatus = 2 OR #ConvStatus = 3) THEN
       #bMove := FALSE;
   END_IF;
   (* выключение перемещения при реверсе*)
   IF #bMoveReverse AND #ConvStatusNext = 0 AND (#ConvStatus = 1 OR #ConvStatus = 3) THEN
       #bMoveReverse := FALSE;
   END_IF;
   (* долгое перемещение*)
   #fbLongMove(IN:=NOT #bStop AND #bMove ,
               PT:=#tLongMove,
               Q=>#bLongMove);
   (* долгое перемещение при реверсе*)
   #fbLongMoveReverse(IN:=NOT #bStop AND #bMoveReverse,
                      PT:=#tLongMove,
                      Q=>#bLongMoveReverse);
   (* включение-выключение перемещения кнопкой*)
   #fbButtMove(CLK:=#bButtMove);
   IF #fbButtMove.Q AND NOT #bMove THEN
       #bOnMove := TRUE;
   END_IF;
   IF #fbButtMove.Q AND #bMove THEN
       #bOffMove := TRUE;
   END_IF;
   IF #bOnMove AND NOT #fbButtMove.Q THEN
       #bMove := TRUE;
       #bOnMove := FALSE;
   END_IF;
   IF #bOffMove AND NOT #fbButtMove.Q THEN
       #bMove := FALSE;
       #bOffMove := FALSE;
   END_IF;
   (* включение-выключение перемещения кнопкой при реверсе*)
   #fbButtMoveReverse(CLK:=#bButtMoveReverse);
   IF #fbButtMoveReverse.Q AND NOT #bMoveReverse THEN
       #bOnMoveReverse := TRUE;
   END_IF;
   IF #fbButtMoveReverse.Q AND #bMoveReverse THEN
       #bOffMoveReverse := TRUE;
   END_IF;
   IF #bOnMoveReverse AND NOT #fbButtMoveReverse.Q THEN
       #bMoveReverse := TRUE;
       #bOnMoveReverse := FALSE;
   END_IF;
   IF #bOffMoveReverse AND NOT #fbButtMoveReverse.Q THEN
       #bMoveReverse := FALSE;
       #bOffMoveReverse := FALSE;
   END_IF;

   IF #bReset THEN
       #bMove := FALSE;
       #bMoveReverse := FALSE;
       #bStartConv := FALSE;
       #bStartConvReverse := FALSE;
   END_IF;

   (* Начальный режим*)
   #fbStartAutomat(CLK:=#bStartAutomat);
   IF #fbStartAutomat.Q AND #bCurtaineUp THEN
       IF NOT #bReverse THEN
           #bStartConv := TRUE;
       ELSE
           #bStartConvReverse := TRUE;
       END_IF;
   END_IF;
   #fbConvBusy1Puls(CLK:=#fbBusy1.ConvBusy);
   #fbConvBusy2Puls(CLK:=#fbBusy2.ConvBusy);
   #fbStartTimer(IN:=#bStartConv,
                 PT:=#tStartTimer);
   #fbStartTimerReverse(IN:=#bStartConvReverse,
                        PT:=#tStartTimer);

   IF (#bFinalConv AND (#ConvStatus = 3 OR #ConvStatus = 2) OR NOT #bFinalConv AND ((#ConvStatus = 3 OR #ConvStatus = 2) AND (#ConvStatusNext = 3 OR #ConvStatusNext = 2)) OR #fbConvBusy2Puls.Q OR #fbStartTimer.Q)
       OR NOT #bStartAutomat
   THEN
       #bStartConv := FALSE;
   END_IF;

   IF (#bStartConvReverse AND (#bFinalConvReverse AND (#ConvStatus = 3 OR #ConvStatus = 1) OR NOT #bFinalConvReverse AND ((#ConvStatus = 3 OR #ConvStatus = 1) AND (#ConvStatusPrev = 3 OR #ConvStatusPrev = 1)) OR #fbConvBusy1Puls.Q OR #fbStartTimerReverse.Q))
       OR NOT #bStartAutomat
   THEN
       #bStartConvReverse := FALSE;
   END_IF;
END_FUNCTION_BLOCK

FUNCTION "FN_IsFree" : Bool   // FC1, SCL
{ S7_Optimized_Access := 'TRUE' }
VERSION : 0.1
   VAR_INPUT
      byConvStatus : Byte;
   END_VAR
BEGIN
   IF #byConvStatus = 0 THEN
       #FN_IsFree := true;
   ELSE
       #FN_IsFree := false;
   END_IF;
   RETURN;
END_FUNCTION

FUNCTION "FN_ConvState" : Byte   // FC2, SCL
{ S7_Optimized_Access := 'TRUE' }
VERSION : 0.1
   VAR_INPUT
      bAuto : Bool;
      bMan : Bool;
      bDrive : Bool;
      bDriveRev : Bool;
      bAlarm : Bool;
   END_VAR
   VAR_TEMP
      byVal : Byte;
   END_VAR
BEGIN
   #byVal := 0;
   IF NOT #bAlarm THEN
       IF #bAuto THEN
           IF #bDrive THEN
               #byVal := 1;
           ELSIF #bDriveRev THEN
               #byVal := 2;
           END_IF;
       ELSE
           IF #bDrive THEN
               #byVal := 3;
           ELSIF #bDriveRev THEN
               #byVal := 4;
           END_IF;
       END_IF;
   ELSE
       #byVal := 5;
   END_IF;
   #FN_ConvState:=#byVal;
   RETURN;
END_FUNCTION

ORGANIZATION_BLOCK "Main"   // OB1, SCL, ProgramCycle
TITLE = "Main Program Sweep (Cycle)"
{ S7_Optimized_Access := 'TRUE' }
VERSION : 0.1
   VAR_INPUT
      Initial_Call : Bool;   // Initial call of this OB
      Remanence : Bool;   // =True, if remanent data are available
   END_VAR
BEGIN
   "FB_SystemTime_DB"();


   "FB_Mode_DB"();
   "FB_Light_DB"(stMode:="FB_Mode_DB".stMode);
   "bMDB_Light_Blue" := "bSDB_Light_Blue" := "FB_Light_DB".bBlue;
   "bMDB_Light_Green" := "bSDB_Light_Green" := "FB_Light_DB".bGreen;
   "bMDB_Light_Yellow" := "bSDB_Light_Yellow" := "FB_Light_DB".bYellow;
   "bMDB_Light_Red" := "bSDB_Light_Red" := "FB_Light_DB".bRed;
   "bMDB_Light_Siren" := "bSDB_Light_Siren" := "FB_Light_DB".bSiren;
END_ORGANIZATION_BLOCK

ORGANIZATION_BLOCK "InboundZone"   // OB123, SCL, ProgramCycle
TITLE = "Main Program Sweep (Cycle)"
{ S7_Optimized_Access := 'TRUE' }
VERSION : 0.1
   VAR_INPUT
      Initial_Call : Bool;   // Initial call of this OB
      Remanence : Bool;   // =True, if remanent data are available
   END_VAR
BEGIN
   "fbConv_001"(wDriveHW_M1:="C1-M1~Data",
                stNext:="fbConv_002".stOut,
                stMode := "FB_Mode_DB".stMode);

   "fbConv_002"(wDriveHW_M1:="C2-M1~Data",
                stNext:="fbConv_003".stOutLine,
                stPrev:="fbConv_001".stOut,
                stMode := "FB_Mode_DB".stMode);

   "fbConv_003"(stNextLine:="fbConv_004".stOut,
                stNextCross:="fbConv_009".stOut,
                stPrevLine:="fbConv_002".stOut,
                stNextLineRev:="fbConv_004".stOutRev,
                stMode:="FB_Mode_DB".stMode);

   "fbConv_004"(stPrev := "fbConv_003".stOutLine,
                stPrevRev:="fbConv_003".stOutLineRev,
                stMode := "FB_Mode_DB".stMode);

   "fbConv_009"(stNext:="fbConv_010".stOut,
                stPrev := "fbConv_003".stOutCross,
                stMode := "FB_Mode_DB".stMode);

   "fbConv_010"(stPrev := "fbConv_009".stOut,
                stMode := "FB_Mode_DB".stMode);
END_ORGANIZATION_BLOCK

ORGANIZATION_BLOCK "Z_EndCycle"   // OB32767, SCL, ProgramCycle
TITLE = "Main Program Sweep (Cycle)"
{ S7_Optimized_Access := 'TRUE' }
VERSION : 0.1
   VAR_INPUT
      Initial_Call : Bool;   // Initial call of this OB
      Remanence : Bool;   // =True, if remanent data are available
   END_VAR
BEGIN
   "bResetAlarm" := FALSE;
END_ORGANIZATION_BLOCK

// folder: FB

FUNCTION_BLOCK "FB_Light"   // FB1, SCL
{ S7_Optimized_Access := 'TRUE' }
VERSION : 0.1
   VAR_INPUT
      stMode : "stModeType";
   END_VAR
   VAR_OUTPUT
      bRed : Bool;
      bYellow : Bool;
      bGreen : Bool;
      bBlue : Bool;
      bSiren : Bool;
   END_VAR
   VAR
      fbTP_Pulse : TP_TIME;
      FB_Pulse_Instance : "FB_Pulse";
      fbTONAlarmSound : TON_TIME;
   END_VAR
   VAR_TEMP
      bPulse : Bool;
   END_VAR
   VAR CONSTANT
      tPulseTime : Time := T#500ms;
      tAlarmSound : Time := T#3s;
   END_VAR
BEGIN
   #bRed := #stMode.bAlarm;
   #bYellow := #stMode.bManual;
   #bGreen := #stMode.bAutomat OR (#stMode.bStartAutomat AND #FB_Pulse_Instance.bPulse);
   #bBlue := #stMode.bReadyToReset;
   #bSiren := #stMode.bAlarm AND #FB_Pulse_Instance.bPulse;

   #fbTONAlarmSound(IN:=#stMode.bAlarm,
                    PT:=#tAlarmSound);


   #FB_Pulse_Instance(bEnable:=#stMode.bStartAutomat OR (#stMode.bAlarm AND NOT #fbTONAlarmSound.Q));
END_FUNCTION_BLOCK

FUNCTION_BLOCK "FB_Mode"   // FB2, SCL
{ S7_Optimized_Access := 'TRUE' }
VERSION : 0.1
   VAR_INPUT
      bAlarm : Bool;   // General system alarm
      bButtAuto : Bool;   // Auto mode button
      bButtStop : Bool;   // Stop mode button
      bButtManu : Bool;   // Manual mode button
      bButtReset : Bool;   // Reset button
      bButtResetAlarm : Bool;   // Reset alarms button
   END_VAR
   VAR_OUTPUT
      stMode : "stModeType";
   END_VAR
BEGIN
   IF #bAlarm THEN
       #stMode.bAutomat := FALSE;
       #stMode.bAlarm := TRUE;
       #stMode.bManual := FALSE;
       #stMode.bAlarm := TRUE;
   ELSIF #bButtReset THEN
       #stMode.bAutomat := FALSE;
       #stMode.bManual := FALSE;
       #stMode.bReset := TRUE;
   ELSIF #bButtStop THEN
       #stMode.bStop := NOT #stMode.bStop;
   ELSIF #bButtManu THEN
       IF NOT #stMode.bAutomat THEN
           #stMode.bManual := NOT #stMode.bManual;
       END_IF;
   ELSIF #bButtAuto THEN
       IF NOT #stMode.bManual THEN
           #stMode.bAutomat := NOT #stMode.bAutomat;
       END_IF;
   ELSIF #bButtResetAlarm THEN
       #stMode.bResetAlarm := TRUE;
   END_IF;

   IF NOT #bButtReset THEN
       #stMode.bReset := FALSE;
   END_IF;

   IF NOT #bButtResetAlarm THEN
       #stMode.bResetAlarm := FALSE;
   END_IF;


   #bButtAuto:= FALSE;
   #bButtStop := FALSE;
   #bButtManu := FALSE;
   #bButtReset := FALSE;
   #bButtResetAlarm := FALSE;
END_FUNCTION_BLOCK

FUNCTION_BLOCK "FB_Pulse"   // FB6, SCL
{ S7_Optimized_Access := 'TRUE' }
VERSION : 0.1
   VAR_INPUT
      bEnable : Bool;
      tPeriod : Time := T#500ms;
   END_VAR
   VAR_OUTPUT
      bPulse : Bool;
   END_VAR
   VAR
      fbTP_Pulse : TP_TIME;
   END_VAR
BEGIN
   IF #bEnable THEN
       #fbTP_Pulse(IN := NOT #fbTP_Pulse.Q,
                   PT := #tPeriod);
       IF #fbTP_Pulse.Q THEN
           #bPulse := NOT #bPulse;
       END_IF;
   ELSE
       #fbTP_Pulse(IN := FALSE,
                   PT := t#0s);
       #bPulse := false;
   END_IF;
END_FUNCTION_BLOCK

FUNCTION_BLOCK "FB_Drive"   // FB14, SCL
{ S7_Optimized_Access := 'TRUE' }
VERSION : 0.1
   VAR_INPUT
      wDriveHW : Hw_Io;
   END_VAR
   VAR_IN_OUT
      stDrive : "stDriveType";
   END_VAR
   VAR
      bWrite : Bool := true;
   END_VAR
   VAR_TEMP
      stDriveIO : "stDriveIOType";
      iResult : Int;
   END_VAR
BEGIN
   //Read IO
   #iResult := DPRD_DAT(LADDR := #wDriveHW, RECORD => #stDriveIO);



   //Write IO
   IF #bWrite THEN
       #iResult := DPWR_DAT(LADDR := #wDriveHW, RECORD := #stDriveIO);
   END_IF;
END_FUNCTION_BLOCK

FUNCTION_BLOCK "FB_SystemTime"   // FB16, SCL
{ S7_Optimized_Access := 'TRUE' }
VERSION : 0.1
   VAR
      dtTime : DTL;
      dtTimeOld : DTL;
      bInit : Bool := true;
      bWrite : Bool;
      fbWriteTimer : TON_TIME;
      iYear : Int;
      iMonth : Int;
      iDay : Int;
      iHour : Int;
      iMinute : Int;
      iSecond : Int;
      iMillisecond : Int;
   END_VAR
   VAR_TEMP
      iResult : Int;
   END_VAR
BEGIN
           #dtTime.YEAR := #iYear;
           #dtTime.MONTH := #iMonth;
           #dtTime.DAY := #iDay;
           #dtTime.HOUR := #iHour;
           #dtTime.MINUTE := #iMinute;
           #dtTime.SECOND := #iSecond;
           IF NOT #bInit THEN
       IF (

           #dtTimeOld.YEAR <> #iYear OR 
           #dtTimeOld.MONTH <> #iMonth OR
           #dtTimeOld.DAY <>  #iDay OR
           #dtTimeOld.HOUR <> #iHour OR
           #dtTimeOld.MINUTE <> #iMinute OR
           #dtTimeOld.SECOND <> #iSecond ) THEN
           #iResult := WR_SYS_T(#dtTime);
           #bWrite := TRUE;
           #dtTimeOld := #dtTime;
       ELSE
           #iResult := RD_SYS_T(#dtTime);
           #dtTimeOld := #dtTime;
       END_IF;
   ELSE
       #iResult := RD_SYS_T(#dtTime);
       #dtTimeOld := #dtTime;
       #bInit := FALSE;
   END_IF;

   #iYear := #dtTime.YEAR;
   #iMonth := #dtTime.MONTH;
   #iDay := #dtTime.DAY;
   #iHour := #dtTime.HOUR;
   #iMinute := #dtTime.MINUTE;
   #iSecond := #dtTime.SECOND;
END_FUNCTION_BLOCK

// folder: FB/Sections

FUNCTION_BLOCK "FB_DirectSection"   // FB3, SCL
{ S7_Optimized_Access := 'TRUE' }
VERSION : 0.1
   VAR_INPUT
      bSens : Bool;   // Sensor free
      stNext : "stOutbound";
      stPrev : "stOutbound";
      tStartTime : Time := T#20s;   // Start mode time limit
      tLongMove : Time := T#40s;   // Long move detection time
      wDriveHW_M1 : Hw_Io;
   END_VAR
   VAR_OUTPUT
      stOut : "stOutbound";
      bLongMove : Bool;   // Long move detected
      byState : Byte;
      bAlarm : Bool;
   END_VAR
   VAR_IN_OUT
      stMode : "stModeType";   // System mode
   END_VAR
   VAR RETAIN
      byConvStatus : Byte;   // Conveyor place status
   END_VAR
   VAR
      bDriveManu : Bool;
      bResManu : Bool;
      bDriveManuReverse : Bool;
      bDriveConv : Bool;
      bOnMove : Bool;
      bOffMove : Bool;
      bDriveConvReverse : Bool;
      bOnMoveReverse : Bool;
      bOffMoveReverse : Bool;
      bStartConv : Bool;
      bStartConvReverse : Bool;
      fbBusy : "FB_Busy1_LAD";
      fbButt : "FB_Button";
      fbButtReverse : "FB_Button";
      fbLongMove : TON_TIME;
      fbLongMoveReverse : TON_TIME;
      fbButtMove : "FB_r_trig";
      fbButtMoveReverse : "FB_r_trig";
      fbStartAutomat : "FB_r_trig";
      fbConvBusy1Puls : "FB_r_trig";
      fbConvBusy2Puls : "FB_r_trig";
      fbStartTimer : TON_TIME;
      fbStartTimerReverse : TON_TIME;
      stDriveM1 : "stDriveType";   // Drive M1 data
      fbR_TRIG_Starting : R_TRIG;   // Starting mode on trigger
      bStarting : Bool;   // Starting mode active
      fbTON_Starting : TON_TIME;   // Starting mode limit timer
      fbDriveM1 : "FB_Drive";
   END_VAR
   // fbBusy.tBusy := T#50ms;
BEGIN
   //Sensors filter
   #fbBusy(bSens := #bSens, Reset := #stMode.bReset);

   //Drive control
   #fbDriveM1(wDriveHW:=#wDriveHW_M1,
              stDrive:=#stDriveM1);

   //Reset
   IF #stMode.bReset THEN
       #byConvStatus := 0;
   END_IF;

   //Starting mode
   #fbR_TRIG_Starting(CLK:=#stMode.bStartAutomat);
   #fbTON_Starting(IN:=#bStarting,
                   PT:=#tStartTime);

   IF #fbR_TRIG_Starting.Q THEN
       IF #fbBusy.ConvBusy THEN
           #byConvStatus:=     2#01000000;
       ELSE
           #byConvStatus := 2#10000010;
       END_IF;
       #bStarting := TRUE;
   END_IF;

   IF #bStarting THEN
       IF NOT #fbR_TRIG_Starting.Q THEN
           IF #fbTON_Starting.Q THEN
               IF #fbBusy.ConvBusy THEN
                   #byConvStatus := 2#11;
               ELSE
                   #byConvStatus := 2#0;
               END_IF;
               #bStarting := FALSE;
           ELSE
               CASE #byConvStatus OF
                   2#01000000:
                       IF #stNext.byConvStatus = 2#10000000 THEN
                           #byConvStatus := 2#01000001;
                       ELSE
                           #byConvStatus := 2#11;
                           #bStarting := FALSE;
                       END_IF;
                   2#01000001:
                       IF NOT #fbBusy.ConvBusy THEN
                           #byConvStatus := 0;
                           #bStarting := FALSE;
                       END_IF;
                   2#10000010:
                       IF #fbBusy.ConvBusy THEN
                           #byConvStatus := 2#11;
                           #bStarting := FALSE;
                       END_IF;
               END_CASE;
           END_IF;
       END_IF;
   ELSE
   //Not starting mode
       IF #stMode.bAutomat AND #bDriveConv THEN
           CASE #byConvStatus OF
               0:
                   IF #stPrev.byConvStatus = 2#01 OR #stPrev.bMove THEN
                       #byConvStatus := 2#10;
                   END_IF;
               2#10:
                   IF #fbBusy.ConvBusy THEN
                       #byConvStatus := 2#11;
                   END_IF;
               2#11:
                   IF #stOut.#bMove THEN
                       #byConvStatus := 2#01;
                   END_IF;
               2#01:
                   IF NOT #fbBusy.ConvBusy THEN
                       #byConvStatus := 2#00;
                   END_IF;
           END_CASE;
       END_IF;
   END_IF;

   //Allow move evaluate
   #stOut.bAllowMove := NOT #stDriveM1.bLock AND NOT #stDriveM1.bAlarm  AND NOT #bLongMove AND (
   //Auto mode
   #stMode.bAutomat AND NOT #fbBusy.ConvBusy AND  #byConvStatus = 0 OR
   //starting mode
   (#bStarting AND #byConvStatus = 2#10000010 AND NOT #fbBusy.ConvBusy)
   );


   //Move evaluate
   #stOut.bMove:=NOT #stDriveM1.bLock AND ((NOT #stOut.#bMove AND #stNext.bAllowMove)OR (#stOut.bMove AND (#byConvStatus = 2#01 OR #byConvStatus = 2#01000001))) AND (
   //Auto mode
   #stMode.bAutomat AND  (#byConvStatus = 2#11 OR #byConvStatus = 2#01)OR
   //starting mode
   (#bStarting AND #byConvStatus = 2#01000001)
   );

   //Drive evaluate
   IF #stMode.bStop OR #stMode.bAlarm THEN
       #bDriveConv := FALSE;
       #bDriveConvReverse := FALSE;
   ELSIF #stMode.bAutomat THEN
       #bDriveConv := NOT #bLongMove AND #stMode.bAutomat AND #stMode.bAutomat AND (
       //inbound
       ((#stPrev.bMove AND (#byConvStatus = 0 OR #byConvStatus = 2#10))OR #byConvStatus = 2#10) OR
       //outbound
       #stOut.bMove);
   ELSIF #stMode.bManual THEN
       ;
   ELSE
       #bDriveConv := FALSE;
       #bDriveConvReverse := FALSE;
   END_IF;

   #stDriveM1.bDrive := #bDriveConv;
   #stDriveM1.bDriveRev := #bDriveConvReverse;

   (* долгое перемещение*)
   #fbLongMove(IN := #bDriveConv AND NOT #bStarting AND (#byConvStatus=2#10 OR #byConvStatus=2#01) AND NOT "bResetAlarm",
               PT := #tLongMove);
   IF #fbLongMove.Q THEN
       #bLongMove := TRUE;
   END_IF;

   //Reset alarms
   IF #stMode.bResetAlarm THEN
       #bLongMove := FALSE;
   END_IF;

   #stOut.bReverse := FALSE;
   #stOut.byConvStatus := #byConvStatus;

   #bAlarm := #stDriveM1.bAlarm OR #bLongMove;

   #byState := "FN_ConvState"(bAuto := #stMode.bAutomat, bMan := #stMode.bManual, bDrive := #stDriveM1.bDrive, bDriveRev := #stDriveM1.bDriveRev, bAlarm := #bAlarm);


   //#bDriveConv := NOT #stMode.bStop AND ((#stMode.bAutomat AND #bMove)OR #bStarting);



   (*
   #bDriveReverse := NOT #bStop AND (#bDriveAutoReverse OR #bDriveConvReverse OR #bDriveManuReverse OR #bStartConvReverse);


   //Manual drive mode
   #bResManu := #bReset OR NOT #bManual;

   #fbButt(bBut:=#bButtManu AND #bManual AND NOT #bDriveManuReverse,
           bRS:= #bResManu,
           bOutB=>#bDriveManu);

   #fbButtReverse(bBut:=#bButtManuReverse AND #bManual  AND NOT #bDriveManu,
                  bRS:=#bResManu,
                  bOutB=>#bDriveManuReverse);

   (*перемещение*)
   (* условия включения перемещения*)
   #bMovePerm := #bAutomat AND #bEnable1 AND #bEnable2 AND (#byConvStatusPrev = 2 OR #byConvStatusPrev = 3) AND #byConvStatus = 0 AND NOT #fbBusyFork.ConvBusy AND NOT #bReverse;
   IF #bMovePerm AND #bCurtaineUp
   THEN
       #bMove := TRUE;
   END_IF;
   (* условия включения обратного перемещения *)
   #bMovePermRev := #bAutomat AND #bEnable3 AND #bEnable4 AND (#byConvStatusNext = 1 OR #byConvStatusNext = 3) AND #byConvStatus = 0 AND NOT #fbBusyFork.ConvBusy AND #bReverse;
   IF #bMovePermRev AND #bCurtaineUp
   THEN
       #bMoveReverse := TRUE;
   END_IF;
   (* включение двигателей *)
   #bDriveConv := NOT #bStop AND #bMove AND NOT (#byConvStatus = 2 OR #byConvStatus = 3);
   #bDrivePrev := NOT #bStop AND #bMove AND NOT (#byConvStatus = 2 OR #byConvStatus = 3) AND NOT (#byConvStatusPrev = 0);
   (* включение двигателей при реверсе*)
   #bDriveConvReverse := NOT #bStop AND #bMoveReverse AND NOT (#byConvStatus = 1 OR #byConvStatus = 3);
   #bDriveNext := NOT #bStop AND #bMoveReverse AND NOT (#byConvStatus = 1 OR #byConvStatus = 3) AND NOT (#byConvStatusNext = 0);
   (* выключение перемещения*)
   IF #bMove AND #byConvStatusPrev = 0 AND (#byConvStatus = 2 OR #byConvStatus = 3) THEN
       #bMove := FALSE;
   END_IF;
   (* выключение перемещения при реверсе*)
   IF #bMoveReverse AND #byConvStatusNext = 0 AND (#byConvStatus = 1 OR #byConvStatus = 3) THEN
       #bMoveReverse := FALSE;
   END_IF;
   (* долгое перемещение при реверсе*)
   #fbLongMoveReverse(IN:=NOT #bStop AND #bMoveReverse,
                      PT:=#tLongMove,
                      Q=>#bLongMoveReverse);
   (* включение-выключение перемещения кнопкой*)
   #fbButtMove(CLK:=#bButtMove);
   IF #fbButtMove.Q AND NOT #bMove THEN
       #bOnMove := TRUE;
   END_IF;
   IF #fbButtMove.Q AND #bMove THEN
       #bOffMove := TRUE;
   END_IF;
   IF #bOnMove AND NOT #fbButtMove.Q THEN
       #bMove := TRUE;
       #bOnMove := FALSE;
   END_IF;
   IF #bOffMove AND NOT #fbButtMove.Q THEN
       #bMove := FALSE;
       #bOffMove := FALSE;
   END_IF;
   (* включение-выключение перемещения кнопкой при реверсе*)
   #fbButtMoveReverse(CLK:=#bButtMoveReverse);
   IF #fbButtMoveReverse.Q AND NOT #bMoveReverse THEN
       #bOnMoveReverse := TRUE;
   END_IF;
   IF #fbButtMoveReverse.Q AND #bMoveReverse THEN
       #bOffMoveReverse := TRUE;
   END_IF;
   IF #bOnMoveReverse AND NOT #fbButtMoveReverse.Q THEN
       #bMoveReverse := TRUE;
       #bOnMoveReverse := FALSE;
   END_IF;
   IF #bOffMoveReverse AND NOT #fbButtMoveReverse.Q THEN
       #bMoveReverse := FALSE;
       #bOffMoveReverse := FALSE;
   END_IF;

   IF #bReset THEN
       #bMove := FALSE;
       #bMoveReverse := FALSE;
       #bStartConv := FALSE;
       #bStartConvReverse := FALSE;
   END_IF;

   (* Начальный режим*)
   #fbStartAutomat(CLK:=#bStartAutomat);
   IF #fbStartAutomat.Q AND #bCurtaineUp THEN
       IF NOT #bReverse THEN
           #bStartConv := TRUE;
       ELSE
           #bStartConvReverse := TRUE;
       END_IF;
   END_IF;
   #fbConvBusy1Puls(CLK:=#fbBusy.ConvBusy);
   #fbConvBusy2Puls(CLK:=#fbBusy2.ConvBusy);
   #fbStartTimer(IN:=#bStartConv,
                 PT:=#tStartTimer);
   #fbStartTimerReverse(IN:=#bStartConvReverse,
                        PT:=#tStartTimer);

   IF (#bFinalConv AND (#byConvStatus = 3 OR #byConvStatus = 2) OR NOT #bFinalConv AND ((#byConvStatus = 3 OR #byConvStatus = 2) AND (#byConvStatusNext = 3 OR #byConvStatusNext = 2)) OR #fbConvBusy2Puls.Q OR #fbStartTimer.Q)
       OR NOT #bStartAutomat
   THEN
       #bStartConv := FALSE;
   END_IF;

   IF (#bStartConvReverse AND (#bFinalConvReverse AND (#byConvStatus = 3 OR #byConvStatus = 1) OR NOT #bFinalConvReverse AND ((#byConvStatus = 3 OR #byConvStatus = 1) AND (#byConvStatusPrev = 3 OR #byConvStatusPrev = 1)) OR #fbConvBusy1Puls.Q OR #fbStartTimerReverse.Q))
       OR NOT #bStartAutomat
   THEN
       #bStartConvReverse := FALSE;
   END_IF;*)
END_FUNCTION_BLOCK

FUNCTION_BLOCK "FB_RotarySection"   // FB15, SCL
{ S7_Optimized_Access := 'TRUE' }
VERSION : 0.1
   VAR_INPUT
      bSens_D1 : Bool;   // Sensor Reverse free
      bSens_D2 : Bool;   // Sensor Direct free
      bSens_D3 : Bool;   // Sensor Overside reverse free
      bSens_D4 : Bool;   // Sensor Overside direct free
      bSens_D5 : Bool;   // Sensor Cross slow pos
      bSens_D6 : Bool;   // Sensor Cross stop pos
      bSens_D7 : Bool;   // Sensor Line slow pos
      bSens_D8 : Bool;   // Sensor Line stop pos
      bSens_Ext : Bool;   // Sensor Overside out free
      bSens_S1 : Bool;   // Sensor Cross stop limit pos
      bSens_S2 : Bool;   // Sensor Line stop limit pos
      stNextLine : "stOutbound";
      stNextLineRev : "stOutbound";
      stNextCross : "stOutbound";
      stPrevLine : "stOutbound";
      tStartTime : Time := T#20s;   // Start mode time limit
      tLongMoveRotary : Time := T#40s;   // Long move detection time
      wDriveHW_M1 : Hw_Io;   // Roller drive
      wDriveHW_M2 : Hw_Io;   // Rotation drive
      bDirectionLine : Bool;   // Move goods to line direction
      bAutoInbound : Bool;   // Auto input selection
   END_VAR
   VAR_OUTPUT
      stOutLine : "stOutbound";
      stOutLineRev : "stOutbound";
      stOutCross : "stOutbound";
      bLongMove : Bool;   // Long move detected
      bSensError : Bool;   // Sensors error
      byRollerState : Byte;
      byRotaryState : Byte;
      bAlarm : Bool;
   END_VAR
   VAR_IN_OUT
      stMode : "stModeType";   // System mode
   END_VAR
   VAR RETAIN
      byConvStatus : Byte;   // Conveyor place status
   END_VAR
   VAR
      bDriveRotary : Bool;
      bDriveRotaryReverse : Bool;
      fbBusy_D3 : "FB_Busy1_LAD";
      fbBusy_D4 : "FB_Busy1_LAD";
      fbBusy_D5 : "FB_Busy1_LAD";
      fbBusy_D6 : "FB_Busy1_LAD";
      fbBusy_D7 : "FB_Busy1_LAD";
      fbBusy_D8 : "FB_Busy1_LAD";
      fbBusy_S1 : "FB_Busy1_LAD";
      fbBusy_S2 : "FB_Busy1_LAD";
      fbBusy_Ext : "FB_Busy1_LAD";
      fbButt : "FB_Button";
      fbButtReverse : "FB_Button";
      fbLongMoveRotary : TON_TIME;
      fbLongMoveReverse : TON_TIME;
      fbButtMove : "FB_r_trig";
      fbButtMoveReverse : "FB_r_trig";
      fbStartAutomat : "FB_r_trig";
      fbConvBusy1Puls : "FB_r_trig";
      fbConvBusy2Puls : "FB_r_trig";
      fbStartTimer : TON_TIME;
      fbStartTimerReverse : TON_TIME;
      stDriveM2 : "stDriveType";   // Drive M1 data
      fbR_TRIG_Starting : R_TRIG;   // Starting mode on trigger
      bStarting : Bool;   // Starting mode active
      fbTON_Starting : TON_TIME;   // Starting mode limit timer
      fbDriveM2 : "FB_Drive";   // Rotation drive
      fbRollerSection : "FB_DirectSectionRev";
      stLine : "stOutbound";
      stCross : "stOutbound";
      byLinedStatus : Byte;
      byCrossedStatus : Byte;
      bLongMoveRotary : Bool;   // Long rotation detected
      bAllowRotation : Bool;   // Allow rotation
      bMiddlePos : Bool;   // Rotary in the middle position
   END_VAR
   VAR_TEMP
      stOutboundDummy : "stOutbound";
      bySensorCount : Byte;
   END_VAR
   // fbBusy_D3.tBusy := T#50ms;
   // fbBusy_D4.tBusy := T#50ms;
   // fbBusy_D5.tBusy := T#50ms;
   // fbBusy_D6.tBusy := T#50ms;
   // fbBusy_D7.tBusy := T#50ms;
   // fbBusy_D8.tBusy := T#50ms;
   // fbBusy_S1.tBusy := T#50ms;
   // fbBusy_S2.tBusy := T#50ms;
   // fbBusy_Ext.tBusy := T#50ms;
BEGIN
   //Sensors filter
   REGION sensor_filter
       #fbBusy_D3(bSens := #bSens_D3,
                  Reset := #stMode.bReset);
       #fbBusy_D4(bSens := #bSens_D4,
                  Reset := #stMode.bReset);
       #fbBusy_D5(bSens := NOT #bSens_D5,
                  Reset := #stMode.bReset);
       #fbBusy_D6(bSens := NOT #bSens_D6,
                  Reset := #stMode.bReset);
       #fbBusy_D7(bSens := NOT #bSens_D7,
                  Reset := #stMode.bReset);
       #fbBusy_D8(bSens := NOT #bSens_D8,
                  Reset := #stMode.bReset);
       #fbBusy_S1(bSens := #bSens_S1,
                  Reset := #stMode.bReset);
       #fbBusy_S2(bSens := #bSens_S2,
                  Reset := #stMode.bReset);
       #fbBusy_Ext(bSens := #bSens_Ext,
                   Reset := #stMode.bReset);
   END_REGION

   REGION sensor_error
       #bySensorCount := BOOL_TO_BYTE(#fbBusy_D5.ConvBusy) + BOOL_TO_BYTE(#fbBusy_D6.ConvBusy) + BOOL_TO_BYTE(#fbBusy_D7.ConvBusy) + BOOL_TO_BYTE(#fbBusy_D8.ConvBusy);
       IF #bySensorCount > 1 OR (#fbBusy_S1.ConvBusy AND #fbBusy_S2.ConvBusy) THEN
           #bSensError := TRUE;
       END_IF;
   END_REGION

   //Roller section control
   #fbRollerSection.stPrev := #stPrevLine;
   #fbRollerSection.stNextRev:= #stNextLineRev;

   #fbRollerSection(bSensDir := #bSens_D2,
                    bSensRev := #bSens_D1,
                    wDriveHW_M1 := #wDriveHW_M1,
                    stMode := #stMode);
   #byConvStatus := #fbRollerSection.byConvStatus;
   #stOutLine.byConvStatus := #fbRollerSection.stOut.byConvStatus;
   #stOutCross.byConvStatus := #fbRollerSection.stOut.byConvStatus;
   #stOutLineRev.byConvStatus := #fbRollerSection.stOut.byConvStatus;

   //Rotary drive control
   #fbDriveM2(wDriveHW:=#wDriveHW_M2,
   stDrive:=#stDriveM2);

   //Reset
   IF #stMode.bReset THEN
       #byConvStatus := 0;
   END_IF;

   //Starting mode
   #fbR_TRIG_Starting(CLK:=#stMode.bStartAutomat);
   #fbTON_Starting(IN:=#bStarting,
                   PT:=#tStartTime);

   IF #fbR_TRIG_Starting.Q THEN
       IF #fbBusy_D3.ConvBusy THEN
           #byConvStatus:=     2#01000000;
       ELSE
           #byConvStatus := 2#10000010;
       END_IF;
       #bStarting := TRUE;
   END_IF;

   IF #bStarting THEN
       IF NOT #fbR_TRIG_Starting.Q THEN
           IF #fbTON_Starting.Q THEN
               IF #fbBusy_D3.ConvBusy THEN
                   #byConvStatus := 2#11;
               ELSE
                   #byConvStatus := 2#0;
               END_IF;
               #bStarting := FALSE;
           ELSE
               CASE #byConvStatus OF
                   2#01000000:
                       IF #stNextLine.byConvStatus = 2#10000000 THEN
                           #byConvStatus := 2#01000001;
                       ELSE
                           #byConvStatus := 2#11;
                           #bStarting := FALSE;
                       END_IF;
                   2#01000001:
                       IF NOT #fbBusy_D3.ConvBusy THEN
                           #byConvStatus := 0;
                           #bStarting := FALSE;
                       END_IF;
                   2#10000010:
                       IF #fbBusy_D3.ConvBusy THEN
                           #byConvStatus := 2#11;
                           #bStarting := FALSE;
                       END_IF;
               END_CASE;
           END_IF;
       END_IF;
   ELSE
   //Not starting mode
       IF #stMode.bAutomat THEN
           IF #fbBusy_D8.ConvBusy THEN
               #byLinedStatus := 2#11;
               #byCrossedStatus := 2#00;
           ELSIF #fbBusy_D6.ConvBusy THEN
               #byLinedStatus := 2#00;
               #byCrossedStatus := 2#11;
           ELSIF #bDriveRotary THEN
               #byLinedStatus := 2#01;
               #byCrossedStatus := 2#10;
           ELSIF #bDriveRotaryReverse THEN
               #byLinedStatus := 2#10;
               #byCrossedStatus := 2#01;
           END_IF;
       END_IF;
   END_IF;

   REGION allow_move
       REGION roller_section
           //Allow move evaluate
           #stOutLine.bAllowMove := #fbRollerSection.stOut.bAllowMove AND #fbBusy_D8.ConvBusy;
           #stOutLineRev.bAllowMove := #fbRollerSection.stOutRev.bAllowMove AND #fbBusy_D8.ConvBusy;
           #stOutCross.bAllowMove:=#fbRollerSection.stOut.bAllowMove AND #fbBusy_D6.ConvBusy;
           #fbRollerSection.stNext.bAllowMove := (#fbBusy_D8.ConvBusy AND #stNextLine.bAllowMove AND #bDirectionLine) OR (#fbBusy_D6.ConvBusy AND #stNextCross.bAllowMove AND NOT #bDirectionLine);
           IF (#fbBusy_D8.ConvBusy) THEN
               #fbRollerSection.stNext.byConvStatus := #stNextLine.byConvStatus;
           ELSIF (#fbBusy_D6.ConvBusy) THEN
               #fbRollerSection.stNext.byConvStatus := #stNextCross.byConvStatus;
           END_IF;
       END_REGION
       REGION rotary_section
           //Rotary allow move evaluate
           #bAllowRotation := NOT #stDriveM2.bLock AND NOT #stDriveM2.bAlarm AND NOT #bLongMoveRotary AND NOT #fbBusy_Ext.ConvBusy AND NOT #fbBusy_D3.ConvBusy AND NOT #fbBusy_D4.ConvBusy;

           #stLine.bAllowMove := #bAllowRotation AND (
           //Auto mode
           (#stMode.bAutomat AND #byLinedStatus <> 2#11)(* OR
           //starting mode
           (#bStarting AND #byConvStatus = 2#10000010 AND NOT #fbBusy_D3.ConvBusy)*)
           );

           #stCross.bAllowMove := #bAllowRotation AND (
           //Auto mode
           (#stMode.bAutomat AND #byCrossedStatus <> 2#11)(* OR
           //starting mode
           (#bStarting AND #byConvStatus = 2#10000010 AND NOT #fbBusy_D3.ConvBusy)*)
           );
       END_REGION
   END_REGION


   REGION move
       REGION roller_section
           #fbRollerSection.stNext.bMove := (#fbBusy_D8.ConvBusy AND #stNextLine.bMove AND #bDirectionLine) OR (#fbBusy_D6.ConvBusy AND #stNextCross.bMove AND NOT #bDirectionLine);
           #stOutCross.bMove := (#fbBusy_D6.ConvBusy AND #fbRollerSection.stOut.bMove AND NOT #bDirectionLine);
           #stOutLine.bMove := (#fbBusy_D8.ConvBusy AND #fbRollerSection.stOut.bMove AND #bDirectionLine);
           //Move evaluate
     (*      #stOutLine.bMove := NOT #stDriveM2.bLock AND ((NOT #stOutLine.#bMove AND #stNextLine.bAllowMove) OR (#stOutLine.bMove AND (#byConvStatus = 2#01 OR #byConvStatus = 2#01000001))) AND (
           //Auto mode
           (#stMode.bAutomat AND (#byConvStatus = 2#11 OR #byConvStatus = 2#01) AND #byLinedStatus = 2#11) OR
           //starting mode
           (#bStarting AND #byConvStatus = 2#01000001)
           );*)
       END_REGION
       REGION rotary_section
           //Move evaluate
           #stLine.bMove := NOT #stDriveM2.bLock AND #stLine.bAllowMove AND (
           //Auto mode
           (#stMode.bAutomat AND ( (NOT #stLine.bMove AND #byConvStatus = 2#00) OR  (#stLine.bMove AND #byLinedStatus<>2#11)))(* OR
           //starting mode
           (#bStarting AND #byConvStatus = 2#01000001)*)
           );

           #stCross.bMove := NOT #stDriveM2.bLock AND #stCross.bAllowMove AND (
           //Auto mode
           (#stMode.bAutomat AND ((NOT #stCross.bMove AND #byConvStatus = 2#11 AND NOT #bDirectionLine) OR (#stCross.bMove AND #byCrossedStatus <> 2#11)))(* OR
           //starting mode
           (#bStarting AND #byConvStatus = 2#01000001)*)
           );
       END_REGION
   END_REGION

   REGION drive
       //Drive evaluate
       IF #stMode.bStop OR #stMode.bAlarm THEN
           #bDriveRotary := FALSE;
           #bDriveRotaryReverse := FALSE;
       ELSIF #stMode.bAutomat THEN
           #bDriveRotary := NOT #bLongMoveRotary AND #stLine.bMove;
           #bDriveRotaryReverse := NOT #bLongMoveRotary AND #stCross.bMove;

           //Drive speed selection
           IF #fbBusy_D6.ConvBusy OR #fbBusy_D8.ConvBusy OR #fbBusy_S1.ConvBusy OR #fbBusy_S2.ConvBusy THEN
               #stDriveM2.bLowSpeed := TRUE;
           ELSE
               IF #bDriveRotary THEN
                   IF #fbBusy_D5.ConvBusy THEN
                       #stDriveM2.bLowSpeed := FALSE;
                   ELSIF #fbBusy_D7.ConvBusy THEN
                       #stDriveM2.bLowSpeed := TRUE;
                   END_IF;
               ELSIF #bDriveRotaryReverse THEN
                   IF #fbBusy_D7.ConvBusy THEN
                       #stDriveM2.bLowSpeed := FALSE;
                   ELSIF #fbBusy_D5.ConvBusy THEN
                       #stDriveM2.bLowSpeed := TRUE;
                   END_IF;
               END_IF;
           END_IF;

       ELSIF #stMode.bManual THEN
           ;
       ELSE
           #bDriveRotary := FALSE;
           #bDriveRotaryReverse := FALSE;
       END_IF;

       #stDriveM2.bDrive := #bDriveRotary;
       #stDriveM2.bDriveRev := #bDriveRotaryReverse;
   END_REGION

   REGION long_move
   (* долгое перемещение*)
       #fbLongMoveRotary(IN := (#stDriveM2.bDrive OR #stDriveM2.bDriveRev) AND NOT #bStarting AND (#stLine.byConvStatus = 2#10 OR #stLine.byConvStatus = 2#01) AND NOT "bResetAlarm",
                         PT := #tLongMoveRotary);
       IF #fbLongMoveRotary.Q THEN
           #bLongMoveRotary := TRUE;
       END_IF;
   END_REGION

   REGION reset_alarms
       //Reset alarms
       IF #stMode.bResetAlarm THEN
           #bLongMoveRotary := FALSE;
           #bSensError := FALSE;
       END_IF;
   END_REGION


   #stOutLine.bReverse := FALSE;
   #stOutLine.byConvStatus := #byConvStatus;

   #stOutLineRev.bReverse := TRUE;
   #stOutLineRev.byConvStatus := #byConvStatus;

   #stOutCross.bReverse := FALSE;
   #stOutCross.byConvStatus := #byConvStatus;

   #byRollerState := #fbRollerSection.byState;
   #byRotaryState := "FN_ConvState"(bAuto := #stMode.bAutomat, bMan := #stMode.bManual, bDrive := #stDriveM2.bDrive, bDriveRev := #stDriveM2.bDriveRev, bAlarm := #stDriveM2.bAlarm OR #bLongMoveRotary);

   #stLine.byConvStatus := #byLinedStatus;

   #stCross.byConvStatus := #byCrossedStatus;

   #bMiddlePos := NOT #fbBusy_D6.ConvBusy AND NOT #fbBusy_D8.ConvBusy;

   //#bDriveConv := NOT #stMode.bStop AND ((#stMode.bAutomat AND #bMove)OR #bStarting);



   (*
   #bDriveReverse := NOT #bStop AND (#bDriveAutoReverse OR #bDriveConvReverse OR #bDriveManuReverse OR #bStartConvReverse);


   //Manual drive mode
   #bResManu := #bReset OR NOT #bManual;

   #fbButt(bBut:=#bButtManu AND #bManual AND NOT #bDriveManuReverse,
           bRS:= #bResManu,
           bOutB=>#bDriveManu);

   #fbButtReverse(bBut:=#bButtManuReverse AND #bManual  AND NOT #bDriveManu,
                  bRS:=#bResManu,
                  bOutB=>#bDriveManuReverse);

   (*перемещение*)
   (* условия включения перемещения*)
   #bMovePerm := #bAutomat AND #bEnable1 AND #bEnable2 AND (#byConvStatusPrev = 2 OR #byConvStatusPrev = 3) AND #byConvStatus = 0 AND NOT #fbBusyFork.ConvBusy AND NOT #bReverse;
   IF #bMovePerm AND #bCurtaineUp
   THEN
       #bMove := TRUE;
   END_IF;
   (* условия включения обратного перемещения *)
   #bMovePermRev := #bAutomat AND #bEnable3 AND #bEnable4 AND (#byConvStatusNext = 1 OR #byConvStatusNext = 3) AND #byConvStatus = 0 AND NOT #fbBusyFork.ConvBusy AND #bReverse;
   IF #bMovePermRev AND #bCurtaineUp
   THEN
       #bMoveReverse := TRUE;
   END_IF;
   (* включение двигателей *)
   #bDriveConv := NOT #bStop AND #bMove AND NOT (#byConvStatus = 2 OR #byConvStatus = 3);
   #bDrivePrev := NOT #bStop AND #bMove AND NOT (#byConvStatus = 2 OR #byConvStatus = 3) AND NOT (#byConvStatusPrev = 0);
   (* включение двигателей при реверсе*)
   #bDriveConvReverse := NOT #bStop AND #bMoveReverse AND NOT (#byConvStatus = 1 OR #byConvStatus = 3);
   #bDriveNext := NOT #bStop AND #bMoveReverse AND NOT (#byConvStatus = 1 OR #byConvStatus = 3) AND NOT (#byConvStatusNext = 0);
   (* выключение перемещения*)
   IF #bMove AND #byConvStatusPrev = 0 AND (#byConvStatus = 2 OR #byConvStatus = 3) THEN
       #bMove := FALSE;
   END_IF;
   (* выключение перемещения при реверсе*)
   IF #bMoveReverse AND #byConvStatusNext = 0 AND (#byConvStatus = 1 OR #byConvStatus = 3) THEN
       #bMoveReverse := FALSE;
   END_IF;
   (* долгое перемещение при реверсе*)
   #fbLongMoveReverse(IN:=NOT #bStop AND #bMoveReverse,
                      PT:=#tLongMove,
                      Q=>#bLongMoveReverse);
   (* включение-выключение перемещения кнопкой*)
   #fbButtMove(CLK:=#bButtMove);
   IF #fbButtMove.Q AND NOT #bMove THEN
       #bOnMove := TRUE;
   END_IF;
   IF #fbButtMove.Q AND #bMove THEN
       #bOffMove := TRUE;
   END_IF;
   IF #bOnMove AND NOT #fbButtMove.Q THEN
       #bMove := TRUE;
       #bOnMove := FALSE;
   END_IF;
   IF #bOffMove AND NOT #fbButtMove.Q THEN
       #bMove := FALSE;
       #bOffMove := FALSE;
   END_IF;
   (* включение-выключение перемещения кнопкой при реверсе*)
   #fbButtMoveReverse(CLK:=#bButtMoveReverse);
   IF #fbButtMoveReverse.Q AND NOT #bMoveReverse THEN
       #bOnMoveReverse := TRUE;
   END_IF;
   IF #fbButtMoveReverse.Q AND #bMoveReverse THEN
       #bOffMoveReverse := TRUE;
   END_IF;
   IF #bOnMoveReverse AND NOT #fbButtMoveReverse.Q THEN
       #bMoveReverse := TRUE;
       #bOnMoveReverse := FALSE;
   END_IF;
   IF #bOffMoveReverse AND NOT #fbButtMoveReverse.Q THEN
       #bMoveReverse := FALSE;
       #bOffMoveReverse := FALSE;
   END_IF;

   IF #bReset THEN
       #bMove := FALSE;
       #bMoveReverse := FALSE;
       #bStartConv := FALSE;
       #bStartConvReverse := FALSE;
   END_IF;

   (* Начальный режим*)
   #fbStartAutomat(CLK:=#bStartAutomat);
   IF #fbStartAutomat.Q AND #bCurtaineUp THEN
       IF NOT #bReverse THEN
           #bStartConv := TRUE;
       ELSE
           #bStartConvReverse := TRUE;
       END_IF;
   END_IF;
   #fbConvBusy1Puls(CLK:=#fbBusy.ConvBusy);
   #fbConvBusy2Puls(CLK:=#fbBusy2.ConvBusy);
   #fbStartTimer(IN:=#bStartConv,
                 PT:=#tStartTimer);
   #fbStartTimerReverse(IN:=#bStartConvReverse,
                        PT:=#tStartTimer);

   IF (#bFinalConv AND (#byConvStatus = 3 OR #byConvStatus = 2) OR NOT #bFinalConv AND ((#byConvStatus = 3 OR #byConvStatus = 2) AND (#byConvStatusNext = 3 OR #byConvStatusNext = 2)) OR #fbConvBusy2Puls.Q OR #fbStartTimer.Q)
       OR NOT #bStartAutomat
   THEN
       #bStartConv := FALSE;
   END_IF;

   IF (#bStartConvReverse AND (#bFinalConvReverse AND (#byConvStatus = 3 OR #byConvStatus = 1) OR NOT #bFinalConvReverse AND ((#byConvStatus = 3 OR #byConvStatus = 1) AND (#byConvStatusPrev = 3 OR #byConvStatusPrev = 1)) OR #fbConvBusy1Puls.Q OR #fbStartTimerReverse.Q))
       OR NOT #bStartAutomat
   THEN
       #bStartConvReverse := FALSE;
   END_IF;*)
END_FUNCTION_BLOCK

FUNCTION_BLOCK "FB_DirectSectionRev"   // FB17, SCL
{ S7_Optimized_Access := 'TRUE' }
VERSION : 0.1
   VAR_INPUT
      bSensDir : Bool;   // Sensor free
      bSensRev : Bool;   // Sensor free
      stNext : "stOutbound";
      stNextRev : "stOutbound";
      stPrev : "stOutbound";
      stPrevRev : "stOutbound";
      tStartTime : Time := T#20s;   // Start mode time limit
      tLongMove : Time := T#40s;   // Long move detection time
      wDriveHW_M1 : Hw_Io;
      bReverse : Bool;
   END_VAR
   VAR_OUTPUT
      stOut : "stOutbound";
      stOutRev : "stOutbound";
      bLongMove : Bool;   // Long move detected
      byState : Byte;
      bAlarm : Bool;
   END_VAR
   VAR_IN_OUT
      stMode : "stModeType";   // System mode
   END_VAR
   VAR RETAIN
      byConvStatus : Byte;   // Conveyor place status
   END_VAR
   VAR
      bDriveManu : Bool;
      bResManu : Bool;
      bDriveManuReverse : Bool;
      bDriveConv : Bool;
      bOnMove : Bool;
      bOffMove : Bool;
      bDriveConvReverse : Bool;
      bOnMoveReverse : Bool;
      bOffMoveReverse : Bool;
      bStartConv : Bool;
      bStartConvReverse : Bool;
      fbBusyDir : "FB_Busy1_LAD";
      fbBusyRev : "FB_Busy1_LAD";
      fbButt : "FB_Button";
      fbButtReverse : "FB_Button";
      fbLongMove : TON_TIME;
      fbLongMoveReverse : TON_TIME;
      fbButtMove : "FB_r_trig";
      fbButtMoveReverse : "FB_r_trig";
      fbStartAutomat : "FB_r_trig";
      fbConvBusy1Puls : "FB_r_trig";
      fbConvBusy2Puls : "FB_r_trig";
      fbStartTimer : TON_TIME;
      fbStartTimerReverse : TON_TIME;
      stDriveM1 : "stDriveType";   // Drive M1 data
      fbR_TRIG_Starting : R_TRIG;   // Starting mode on trigger
      bStarting : Bool;   // Starting mode active
      fbTON_Starting : TON_TIME;   // Starting mode limit timer
      fbDriveM1 : "FB_Drive";
   END_VAR
   // fbBusyDir.tBusy := T#50ms;
   // fbBusyRev.tBusy := T#50ms;
BEGIN
   //Sensors filter
   #fbBusyDir(bSens := #bSensDir, Reset := #stMode.bReset);
   #fbBusyRev(bSens := #bSensRev,
           Reset := #stMode.bReset);

   //Drive control
   #fbDriveM1(wDriveHW:=#wDriveHW_M1,
              stDrive:=#stDriveM1);

   //Reset
   IF #stMode.bReset THEN
       #byConvStatus := 0;
   END_IF;

   //Starting mode
   #fbR_TRIG_Starting(CLK:=#stMode.bStartAutomat);
   #fbTON_Starting(IN := #bStarting,
                   PT := #tStartTime);

   IF #fbR_TRIG_Starting.Q THEN
       IF #fbBusyDir.ConvBusy THEN
           #byConvStatus:=     2#01000000;
       ELSE
           #byConvStatus := 2#10000010;
       END_IF;
       #bStarting := TRUE;
   END_IF;

   IF #bStarting THEN
       IF NOT #fbR_TRIG_Starting.Q THEN
           IF #fbTON_Starting.Q THEN
               IF #fbBusyDir.ConvBusy THEN
                   #byConvStatus := 2#11;
               ELSE
                   #byConvStatus := 2#0;
               END_IF;
               #bStarting := FALSE;
           ELSE
               CASE #byConvStatus OF
                   2#01000000:
                       IF #stNext.byConvStatus = 2#10000000 THEN
                           #byConvStatus := 2#01000001;
                       ELSE
                           #byConvStatus := 2#11;
                           #bStarting := FALSE;
                       END_IF;
                   2#01000001:
                       IF NOT #fbBusyDir.ConvBusy THEN
                           #byConvStatus := 0;
                           #bStarting := FALSE;
                       END_IF;
                   2#10000010:
                       IF #fbBusyDir.ConvBusy THEN
                           #byConvStatus := 2#11;
                           #bStarting := FALSE;
                       END_IF;
               END_CASE;
           END_IF;
       END_IF;
   ELSE
   //Not starting mode
       IF #stMode.bAutomat THEN
           IF #bDriveConv THEN
               CASE #byConvStatus OF
                   0:
                       IF #stPrev.byConvStatus = 2#01 OR #stPrev.bMove THEN
                           #byConvStatus := 2#10;
                       END_IF;
                   2#10:
                       IF #fbBusyDir.ConvBusy THEN
                           #byConvStatus := 2#11;
                       END_IF;
                   2#11:
                       IF #stOut.#bMove THEN
                           #byConvStatus := 2#01;
                       END_IF;
                   2#01:
                       IF NOT #fbBusyDir.ConvBusy THEN
                           #byConvStatus := 2#00;
                       END_IF;
               END_CASE;
           ELSIF #bDriveConvReverse THEN
               CASE #byConvStatus OF
                   0:
                       IF #stNextRev.byConvStatus = 2#10 OR #stNextRev.bMove THEN
                           #byConvStatus := 2#01;
                       END_IF;
                   2#01:
                       IF #fbBusyRev.ConvBusy THEN
                           #byConvStatus := 2#11;
                       END_IF;
                   2#11:
                       IF #stOutRev.#bMove THEN
                           #byConvStatus := 2#10;
                       END_IF;
                   2#10:
                       IF NOT #fbBusyRev.ConvBusy THEN
                           #byConvStatus := 2#00;
                       END_IF;
               END_CASE;
           END_IF;
       END_IF;
   END_IF;

   //Allow move direct evaluate
   //Direct
   #stOut.bAllowMove := NOT #bReverse AND NOT #stDriveM1.bLock AND NOT #stDriveM1.bAlarm  AND NOT #bLongMove AND (
   //Auto mode
   #stMode.bAutomat AND NOT #fbBusyDir.ConvBusy AND  #byConvStatus = 0 OR
   //starting mode
   (#bStarting AND #byConvStatus = 2#10000010 AND NOT #fbBusyDir.ConvBusy)
   );

   //Reverse
   #stOutRev.bAllowMove := #bReverse AND NOT #stDriveM1.bLock AND NOT #stDriveM1.bAlarm AND NOT #bLongMove AND (
   //Auto mode
   #stMode.bAutomat AND NOT #fbBusyRev.ConvBusy AND #byConvStatus = 0 OR
   //starting mode
   (#bStarting AND #byConvStatus = 2#10000001 AND NOT #fbBusyRev.ConvBusy)
   );

   //Move evaluate
   #stOut.bMove:=NOT #bReverse  AND NOT #stDriveM1.bLock AND ((NOT #stOut.#bMove AND #stNext.bAllowMove)OR (#stOut.bMove AND (#byConvStatus = 2#01 OR #byConvStatus = 2#01000001))) AND (
   //Auto mode
   #stMode.bAutomat AND  (#byConvStatus = 2#11 OR #byConvStatus = 2#01)OR
   //starting mode
   (#bStarting AND #byConvStatus = 2#01000001)
   );

   //Move evaluate
   #stOutRev.bMove :=#bReverse AND  NOT #stDriveM1.bLock AND ((NOT #stOutRev.#bMove AND #stPrevRev.bAllowMove) OR (#stOutRev.bMove AND (#byConvStatus = 2#10 OR #byConvStatus = 2#01000010))) AND (
   //Auto mode
   #stMode.bAutomat AND (#byConvStatus = 2#11 OR #byConvStatus = 2#10) OR
   //starting mode
   (#bStarting AND #byConvStatus = 2#01000001)
   );


   //Drive evaluate
   IF #stMode.bStop OR #stMode.bAlarm THEN
       #bDriveConv := FALSE;
       #bDriveConvReverse := FALSE;
   ELSIF #stMode.bAutomat THEN
       #bDriveConv := NOT #bReverse AND NOT #bLongMove AND (
       //inbound
       ((#stPrev.bMove AND (#byConvStatus = 0 OR #byConvStatus = 2#10))OR #byConvStatus = 2#10) OR
       //outbound
       #stOut.bMove);

       #bDriveConvReverse := #bReverse AND NOT #bLongMove AND (
       //inbound
       ((#stNextRev.bMove AND (#byConvStatus = 0 OR #byConvStatus = 2#01)) OR #byConvStatus = 2#01) OR
       //outbound
       #stOutRev.bMove);

   ELSIF #stMode.bManual THEN
       ;
   ELSE
       #bDriveConv := FALSE;
       #bDriveConvReverse := FALSE;
   END_IF;

   #stDriveM1.bDrive := #bDriveConv;
   #stDriveM1.bDriveRev := #bDriveConvReverse;

   (* долгое перемещение*)
   #fbLongMove(IN := (#bDriveConv OR #bDriveConvReverse) AND NOT #bStarting AND (#byConvStatus=2#10 OR #byConvStatus=2#01) AND NOT "bResetAlarm",
               PT := #tLongMove);
   IF #fbLongMove.Q THEN
       #bLongMove := TRUE;
   END_IF;

   //Reset alarms
   IF #stMode.bResetAlarm THEN
       #bLongMove := FALSE;
   END_IF;

   #stOut.bReverse := FALSE;
   #stOut.byConvStatus := #byConvStatus;

   #stOutRev.bReverse := TRUE;
   #stOutRev.byConvStatus := #byConvStatus;


   #bAlarm := #stDriveM1.bAlarm OR #bLongMove;

   #byState := "FN_ConvState"(bAuto := #stMode.bAutomat, bMan := #stMode.bManual, bDrive := #stDriveM1.bDrive, bDriveRev := #stDriveM1.bDriveRev, bAlarm := #bAlarm);


   //#bDriveConv := NOT #stMode.bStop AND ((#stMode.bAutomat AND #bMove)OR #bStarting);



   (*
   #bDriveReverse := NOT #bStop AND (#bDriveAutoReverse OR #bDriveConvReverse OR #bDriveManuReverse OR #bStartConvReverse);


   //Manual drive mode
   #bResManu := #bReset OR NOT #bManual;

   #fbButt(bBut:=#bButtManu AND #bManual AND NOT #bDriveManuReverse,
           bRS:= #bResManu,
           bOutB=>#bDriveManu);

   #fbButtReverse(bBut:=#bButtManuReverse AND #bManual  AND NOT #bDriveManu,
                  bRS:=#bResManu,
                  bOutB=>#bDriveManuReverse);

   (*перемещение*)
   (* условия включения перемещения*)
   #bMovePerm := #bAutomat AND #bEnable1 AND #bEnable2 AND (#byConvStatusPrev = 2 OR #byConvStatusPrev = 3) AND #byConvStatus = 0 AND NOT #fbBusyFork.ConvBusy AND NOT #bReverse;
   IF #bMovePerm AND #bCurtaineUp
   THEN
       #bMove := TRUE;
   END_IF;
   (* условия включения обратного перемещения *)
   #bMovePermRev := #bAutomat AND #bEnable3 AND #bEnable4 AND (#byConvStatusNext = 1 OR #byConvStatusNext = 3) AND #byConvStatus = 0 AND NOT #fbBusyFork.ConvBusy AND #bReverse;
   IF #bMovePermRev AND #bCurtaineUp
   THEN
       #bMoveReverse := TRUE;
   END_IF;
   (* включение двигателей *)
   #bDriveConv := NOT #bStop AND #bMove AND NOT (#byConvStatus = 2 OR #byConvStatus = 3);
   #bDrivePrev := NOT #bStop AND #bMove AND NOT (#byConvStatus = 2 OR #byConvStatus = 3) AND NOT (#byConvStatusPrev = 0);
   (* включение двигателей при реверсе*)
   #bDriveConvReverse := NOT #bStop AND #bMoveReverse AND NOT (#byConvStatus = 1 OR #byConvStatus = 3);
   #bDriveNext := NOT #bStop AND #bMoveReverse AND NOT (#byConvStatus = 1 OR #byConvStatus = 3) AND NOT (#byConvStatusNext = 0);
   (* выключение перемещения*)
   IF #bMove AND #byConvStatusPrev = 0 AND (#byConvStatus = 2 OR #byConvStatus = 3) THEN
       #bMove := FALSE;
   END_IF;
   (* выключение перемещения при реверсе*)
   IF #bMoveReverse AND #byConvStatusNext = 0 AND (#byConvStatus = 1 OR #byConvStatus = 3) THEN
       #bMoveReverse := FALSE;
   END_IF;
   (* долгое перемещение при реверсе*)
   #fbLongMoveReverse(IN:=NOT #bStop AND #bMoveReverse,
                      PT:=#tLongMove,
                      Q=>#bLongMoveReverse);
   (* включение-выключение перемещения кнопкой*)
   #fbButtMove(CLK:=#bButtMove);
   IF #fbButtMove.Q AND NOT #bMove THEN
       #bOnMove := TRUE;
   END_IF;
   IF #fbButtMove.Q AND #bMove THEN
       #bOffMove := TRUE;
   END_IF;
   IF #bOnMove AND NOT #fbButtMove.Q THEN
       #bMove := TRUE;
       #bOnMove := FALSE;
   END_IF;
   IF #bOffMove AND NOT #fbButtMove.Q THEN
       #bMove := FALSE;
       #bOffMove := FALSE;
   END_IF;
   (* включение-выключение перемещения кнопкой при реверсе*)
   #fbButtMoveReverse(CLK:=#bButtMoveReverse);
   IF #fbButtMoveReverse.Q AND NOT #bMoveReverse THEN
       #bOnMoveReverse := TRUE;
   END_IF;
   IF #fbButtMoveReverse.Q AND #bMoveReverse THEN
       #bOffMoveReverse := TRUE;
   END_IF;
   IF #bOnMoveReverse AND NOT #fbButtMoveReverse.Q THEN
       #bMoveReverse := TRUE;
       #bOnMoveReverse := FALSE;
   END_IF;
   IF #bOffMoveReverse AND NOT #fbButtMoveReverse.Q THEN
       #bMoveReverse := FALSE;
       #bOffMoveReverse := FALSE;
   END_IF;

   IF #bReset THEN
       #bMove := FALSE;
       #bMoveReverse := FALSE;
       #bStartConv := FALSE;
       #bStartConvReverse := FALSE;
   END_IF;

   (* Начальный режим*)
   #fbStartAutomat(CLK:=#bStartAutomat);
   IF #fbStartAutomat.Q AND #bCurtaineUp THEN
       IF NOT #bReverse THEN
           #bStartConv := TRUE;
       ELSE
           #bStartConvReverse := TRUE;
       END_IF;
   END_IF;
   #fbConvBusy1Puls(CLK:=#fbBusy.ConvBusy);
   #fbConvBusy2Puls(CLK:=#fbBusy2.ConvBusy);
   #fbStartTimer(IN:=#bStartConv,
                 PT:=#tStartTimer);
   #fbStartTimerReverse(IN:=#bStartConvReverse,
                        PT:=#tStartTimer);

   IF (#bFinalConv AND (#byConvStatus = 3 OR #byConvStatus = 2) OR NOT #bFinalConv AND ((#byConvStatus = 3 OR #byConvStatus = 2) AND (#byConvStatusNext = 3 OR #byConvStatusNext = 2)) OR #fbConvBusy2Puls.Q OR #fbStartTimer.Q)
       OR NOT #bStartAutomat
   THEN
       #bStartConv := FALSE;
   END_IF;

   IF (#bStartConvReverse AND (#bFinalConvReverse AND (#byConvStatus = 3 OR #byConvStatus = 1) OR NOT #bFinalConvReverse AND ((#byConvStatus = 3 OR #byConvStatus = 1) AND (#byConvStatusPrev = 3 OR #byConvStatusPrev = 1)) OR #fbConvBusy1Puls.Q OR #fbStartTimerReverse.Q))
       OR NOT #bStartAutomat
   THEN
       #bStartConvReverse := FALSE;
   END_IF;*)
END_FUNCTION_BLOCK

FUNCTION_BLOCK "FB_TransferSection"   // FB18, SCL
{ S7_Optimized_Access := 'TRUE' }
VERSION : 0.1
   VAR_INPUT
      bSens_D1 : Bool;   // Sensor Reverse free
      bSens_D2 : Bool;   // Sensor Direct free
      bSens_D3 : Bool;   // Sensor Overside reverse free
      bSens_D4 : Bool;   // Sensor Overside direct free
      bSens_D5 : Bool;   // Sensor Cross slow pos
      bSens_D6 : Bool;   // Sensor Cross stop pos
      bSens_D7 : Bool;   // Sensor Line slow pos
      bSens_D8 : Bool;   // Sensor Line stop pos
      bSens_S1 : Bool;   // Sensor Cross stop limit pos
      bSens_S2 : Bool;   // Sensor Line stop limit pos
      stNextLine : "stOutbound";
      stNextCross : "stOutbound";
      stPrevLine : "stOutbound";
      stPrevLineRev : "stOutbound";
      tStartTime : Time := T#20s;   // Start mode time limit
      tLongMove : Time := T#40s;   // Long move detection time
      wDriveHW_M1 : Hw_Io;   // Roller drive
      wDriveHW_M2 : Hw_Io;   // Rotation drive
      bDirectionLine : Hw_Io;
   END_VAR
   VAR_OUTPUT
      stOutLine : "stOutbound";
      stOutCross : "stOutbound";
      bLongMove : Bool;   // Long move detected
   END_VAR
   VAR_IN_OUT
      stMode : "stModeType";   // System mode
   END_VAR
   VAR RETAIN
      byConvStatus : Byte;   // Conveyor place status
   END_VAR
   VAR
      bDriveManu : Bool;
      bResManu : Bool;
      bDriveManuReverse : Bool;
      bDriveConv : Bool;
      bOnMove : Bool;
      bOffMove : Bool;
      bDriveConvReverse : Bool;
      bOnMoveReverse : Bool;
      bOffMoveReverse : Bool;
      bStartConv : Bool;
      bStartConvReverse : Bool;
      fbBusy_D3 : "FB_Busy1_LAD";
      fbBusy_D4 : "FB_Busy1_LAD";
      fbBusy_D5 : "FB_Busy1_LAD";
      fbBusy_D6 : "FB_Busy1_LAD";
      fbBusy_D7 : "FB_Busy1_LAD";
      fbBusy_D8 : "FB_Busy1_LAD";
      fbBusy_S1 : "FB_Busy1_LAD";
      fbBusy_S2 : "FB_Busy1_LAD";
      fbButt : "FB_Button";
      fbButtReverse : "FB_Button";
      fbLongMove : TON_TIME;
      fbLongMoveReverse : TON_TIME;
      fbButtMove : "FB_r_trig";
      fbButtMoveReverse : "FB_r_trig";
      fbStartAutomat : "FB_r_trig";
      fbConvBusy1Puls : "FB_r_trig";
      fbConvBusy2Puls : "FB_r_trig";
      fbStartTimer : TON_TIME;
      fbStartTimerReverse : TON_TIME;
      stDriveM1 : "stDriveType";   // Drive M1 data
      fbR_TRIG_Starting : R_TRIG;   // Starting mode on trigger
      bStarting : Bool;   // Starting mode active
      fbTON_Starting : TON_TIME;   // Starting mode limit timer
      fbDriveM1 : "FB_Drive";   // Roller drive
      fbDriveM2 : "FB_Drive";   // Rotation drive
      FB_DirectSectionRev_Instance : "FB_DirectSectionRev";
   END_VAR
   // fbBusy_D3.tBusy := T#50ms;
   // fbBusy_D4.tBusy := T#50ms;
   // fbBusy_D5.tBusy := T#50ms;
   // fbBusy_D6.tBusy := T#50ms;
   // fbBusy_D7.tBusy := T#50ms;
   // fbBusy_D8.tBusy := T#50ms;
   // fbBusy_S1.tBusy := T#50ms;
   // fbBusy_S2.tBusy := T#50ms;
BEGIN
   //Sensors filter
   #fbBusy_D3(bSens := #bSens_D3,
              Reset := #stMode.bReset);
   #fbBusy_D4(bSens := #bSens_D4,
              Reset := #stMode.bReset);
   #fbBusy_D5(bSens := #bSens_D5,
              Reset := #stMode.bReset);
   #fbBusy_D6(bSens := #bSens_D6,
              Reset := #stMode.bReset);
   #fbBusy_D7(bSens := #bSens_D7,
              Reset := #stMode.bReset);
   #fbBusy_D8(bSens := #bSens_D8,
              Reset := #stMode.bReset);
   #fbBusy_S1(bSens := #bSens_S1,
              Reset := #stMode.bReset);
   #fbBusy_S2(bSens := #bSens_S2,
              Reset := #stMode.bReset);


   //Drive control
   //#fbDriveM1(wDriveHW:=#wDriveHW_M1,
   //stDrive:=#stDriveM1);

   //Roller section control
   #FB_DirectSectionRev_Instance(bSensDir:=#bSens_D1,
                                 bSensRev:=#bSens_D2,
                                 wDriveHW_M1:=#wDriveHW_M1,
                                 stMode:=#stMode);



   //Reset
   IF #stMode.bReset THEN
       #byConvStatus := 0;
   END_IF;

   //Starting mode
   #fbR_TRIG_Starting(CLK:=#stMode.bStartAutomat);
   #fbTON_Starting(IN:=#bStarting,
                   PT:=#tStartTime);

   IF #fbR_TRIG_Starting.Q THEN
       IF #fbBusy_D3.ConvBusy THEN
           #byConvStatus:=     2#01000000;
       ELSE
           #byConvStatus := 2#10000010;
       END_IF;
       #bStarting := TRUE;
   END_IF;

   IF #bStarting THEN
       IF NOT #fbR_TRIG_Starting.Q THEN
           IF #fbTON_Starting.Q THEN
               IF #fbBusy_D3.ConvBusy THEN
                   #byConvStatus := 2#11;
               ELSE
                   #byConvStatus := 2#0;
               END_IF;
               #bStarting := FALSE;
           ELSE
               CASE #byConvStatus OF
                   2#01000000:
                       IF #stNextLine.byConvStatus = 2#10000000 THEN
                           #byConvStatus := 2#01000001;
                       ELSE
                           #byConvStatus := 2#11;
                           #bStarting := FALSE;
                       END_IF;
                   2#01000001:
                       IF NOT #fbBusy_D3.ConvBusy THEN
                           #byConvStatus := 0;
                           #bStarting := FALSE;
                       END_IF;
                   2#10000010:
                       IF #fbBusy_D3.ConvBusy THEN
                           #byConvStatus := 2#11;
                           #bStarting := FALSE;
                       END_IF;
               END_CASE;
           END_IF;
       END_IF;
   ELSE
   //Not starting mode
       IF #stMode.bAutomat AND #bDriveConv THEN
           CASE #byConvStatus OF
               0:
                   IF #stPrevLine.byConvStatus = 2#01 OR #stPrevLine.bMove THEN
                       #byConvStatus := 2#10;
                   END_IF;
               2#10:
                   IF #fbBusy_D3.ConvBusy THEN
                       #byConvStatus := 2#11;
                   END_IF;
               2#11:
                   IF #stOutLine.#bMove THEN
                       #byConvStatus := 2#01;
                   END_IF;
               2#01:
                   IF NOT #fbBusy_D3.ConvBusy THEN
                       #byConvStatus := 2#00;
                   END_IF;
           END_CASE;
       END_IF;
   END_IF;

   //Allow move evaluate
   #stOutLine.bAllowMove := NOT #stDriveM1.bLock AND NOT #stDriveM1.bAlarm  AND NOT #bLongMove AND (
   //Auto mode
   #stMode.bAutomat AND NOT #fbBusy_D3.ConvBusy AND  #byConvStatus = 0 OR
   //starting mode
   (#bStarting AND #byConvStatus = 2#10000010 AND NOT #fbBusy_D3.ConvBusy)
   );


   //Move evaluate
   #stOutLine.bMove:=NOT #stDriveM1.bLock AND ((NOT #stOutLine.#bMove AND #stNextLine.bAllowMove)OR (#stOutLine.bMove AND (#byConvStatus = 2#01 OR #byConvStatus = 2#01000001))) AND (
   //Auto mode
   #stMode.bAutomat AND  (#byConvStatus = 2#11 OR #byConvStatus = 2#01)OR
   //starting mode
   (#bStarting AND #byConvStatus = 2#01000001)
   );

   //Drive evaluate
   IF #stMode.bStop OR #stMode.bAlarm THEN
       #bDriveConv := FALSE;
       #bDriveConvReverse := FALSE;
   ELSIF #stMode.bAutomat THEN
       #bDriveConv := NOT #bLongMove AND #stMode.bAutomat AND #stMode.bAutomat AND (
       //inbound
       ((#stPrevLine.bMove AND (#byConvStatus = 0 OR #byConvStatus = 2#10))OR #byConvStatus = 2#10) OR
       //outbound
       #stOutLine.bMove);
   ELSIF #stMode.bManual THEN
       ;
   ELSE
       #bDriveConv := FALSE;
       #bDriveConvReverse := FALSE;
   END_IF;

   #stDriveM1.bDrive := #bDriveConv;
   #stDriveM1.bDriveRev := #bDriveConvReverse;

   (* долгое перемещение*)
   #fbLongMove(IN := #bDriveConv AND NOT #bStarting AND (#byConvStatus=2#10 OR #byConvStatus=2#01) AND NOT "bResetAlarm",
               PT := #tLongMove);
   IF #fbLongMove.Q THEN
       #bLongMove := TRUE;
   END_IF;

   //Reset alarms
   IF #stMode.bResetAlarm THEN
       #bLongMove := FALSE;
   END_IF;

   #stOutLine.bReverse := FALSE;
   #stOutLine.byConvStatus := #byConvStatus;






   //#bDriveConv := NOT #stMode.bStop AND ((#stMode.bAutomat AND #bMove)OR #bStarting);



   (*
   #bDriveReverse := NOT #bStop AND (#bDriveAutoReverse OR #bDriveConvReverse OR #bDriveManuReverse OR #bStartConvReverse);


   //Manual drive mode
   #bResManu := #bReset OR NOT #bManual;

   #fbButt(bBut:=#bButtManu AND #bManual AND NOT #bDriveManuReverse,
           bRS:= #bResManu,
           bOutB=>#bDriveManu);

   #fbButtReverse(bBut:=#bButtManuReverse AND #bManual  AND NOT #bDriveManu,
                  bRS:=#bResManu,
                  bOutB=>#bDriveManuReverse);

   (*перемещение*)
   (* условия включения перемещения*)
   #bMovePerm := #bAutomat AND #bEnable1 AND #bEnable2 AND (#byConvStatusPrev = 2 OR #byConvStatusPrev = 3) AND #byConvStatus = 0 AND NOT #fbBusyFork.ConvBusy AND NOT #bReverse;
   IF #bMovePerm AND #bCurtaineUp
   THEN
       #bMove := TRUE;
   END_IF;
   (* условия включения обратного перемещения *)
   #bMovePermRev := #bAutomat AND #bEnable3 AND #bEnable4 AND (#byConvStatusNext = 1 OR #byConvStatusNext = 3) AND #byConvStatus = 0 AND NOT #fbBusyFork.ConvBusy AND #bReverse;
   IF #bMovePermRev AND #bCurtaineUp
   THEN
       #bMoveReverse := TRUE;
   END_IF;
   (* включение двигателей *)
   #bDriveConv := NOT #bStop AND #bMove AND NOT (#byConvStatus = 2 OR #byConvStatus = 3);
   #bDrivePrev := NOT #bStop AND #bMove AND NOT (#byConvStatus = 2 OR #byConvStatus = 3) AND NOT (#byConvStatusPrev = 0);
   (* включение двигателей при реверсе*)
   #bDriveConvReverse := NOT #bStop AND #bMoveReverse AND NOT (#byConvStatus = 1 OR #byConvStatus = 3);
   #bDriveNext := NOT #bStop AND #bMoveReverse AND NOT (#byConvStatus = 1 OR #byConvStatus = 3) AND NOT (#byConvStatusNext = 0);
   (* выключение перемещения*)
   IF #bMove AND #byConvStatusPrev = 0 AND (#byConvStatus = 2 OR #byConvStatus = 3) THEN
       #bMove := FALSE;
   END_IF;
   (* выключение перемещения при реверсе*)
   IF #bMoveReverse AND #byConvStatusNext = 0 AND (#byConvStatus = 1 OR #byConvStatus = 3) THEN
       #bMoveReverse := FALSE;
   END_IF;
   (* долгое перемещение при реверсе*)
   #fbLongMoveReverse(IN:=NOT #bStop AND #bMoveReverse,
                      PT:=#tLongMove,
                      Q=>#bLongMoveReverse);
   (* включение-выключение перемещения кнопкой*)
   #fbButtMove(CLK:=#bButtMove);
   IF #fbButtMove.Q AND NOT #bMove THEN
       #bOnMove := TRUE;
   END_IF;
   IF #fbButtMove.Q AND #bMove THEN
       #bOffMove := TRUE;
   END_IF;
   IF #bOnMove AND NOT #fbButtMove.Q THEN
       #bMove := TRUE;
       #bOnMove := FALSE;
   END_IF;
   IF #bOffMove AND NOT #fbButtMove.Q THEN
       #bMove := FALSE;
       #bOffMove := FALSE;
   END_IF;
   (* включение-выключение перемещения кнопкой при реверсе*)
   #fbButtMoveReverse(CLK:=#bButtMoveReverse);
   IF #fbButtMoveReverse.Q AND NOT #bMoveReverse THEN
       #bOnMoveReverse := TRUE;
   END_IF;
   IF #fbButtMoveReverse.Q AND #bMoveReverse THEN
       #bOffMoveReverse := TRUE;
   END_IF;
   IF #bOnMoveReverse AND NOT #fbButtMoveReverse.Q THEN
       #bMoveReverse := TRUE;
       #bOnMoveReverse := FALSE;
   END_IF;
   IF #bOffMoveReverse AND NOT #fbButtMoveReverse.Q THEN
       #bMoveReverse := FALSE;
       #bOffMoveReverse := FALSE;
   END_IF;

   IF #bReset THEN
       #bMove := FALSE;
       #bMoveReverse := FALSE;
       #bStartConv := FALSE;
       #bStartConvReverse := FALSE;
   END_IF;

   (* Начальный режим*)
   #fbStartAutomat(CLK:=#bStartAutomat);
   IF #fbStartAutomat.Q AND #bCurtaineUp THEN
       IF NOT #bReverse THEN
           #bStartConv := TRUE;
       ELSE
           #bStartConvReverse := TRUE;
       END_IF;
   END_IF;
   #fbConvBusy1Puls(CLK:=#fbBusy.ConvBusy);
   #fbConvBusy2Puls(CLK:=#fbBusy2.ConvBusy);
   #fbStartTimer(IN:=#bStartConv,
                 PT:=#tStartTimer);
   #fbStartTimerReverse(IN:=#bStartConvReverse,
                        PT:=#tStartTimer);

   IF (#bFinalConv AND (#byConvStatus = 3 OR #byConvStatus = 2) OR NOT #bFinalConv AND ((#byConvStatus = 3 OR #byConvStatus = 2) AND (#byConvStatusNext = 3 OR #byConvStatusNext = 2)) OR #fbConvBusy2Puls.Q OR #fbStartTimer.Q)
       OR NOT #bStartAutomat
   THEN
       #bStartConv := FALSE;
   END_IF;

   IF (#bStartConvReverse AND (#bFinalConvReverse AND (#byConvStatus = 3 OR #byConvStatus = 1) OR NOT #bFinalConvReverse AND ((#byConvStatus = 3 OR #byConvStatus = 1) AND (#byConvStatusPrev = 3 OR #byConvStatusPrev = 1)) OR #fbConvBusy1Puls.Q OR #fbStartTimerReverse.Q))
       OR NOT #bStartAutomat
   THEN
       #bStartConvReverse := FALSE;
   END_IF;*)
END_FUNCTION_BLOCK

// folder: FB_OLD

FUNCTION_BLOCK "FB_Busy1_LAD"   // FB8, LAD
{ S7_Optimized_Access := 'FALSE' }
VERSION : 0.1
// Фильтр для оптического датчика
   VAR_INPUT
      bSens : Bool;
      tBusy : Time;
      tFree : Time;
      Reset : Bool;
   END_VAR
   VAR_OUTPUT
      ConvBusy : Bool;
   END_VAR
   VAR
      bConvBusy1 : Bool := false;
      bNotConvBusy : Bool;
      bTest : Bool;
      Timer1 : TON_TIME;
      Timer2 : TON_TIME;
      IEC_Timer_0_Instance : TON_TIME;
   END_VAR
BEGIN

REGION Network 1
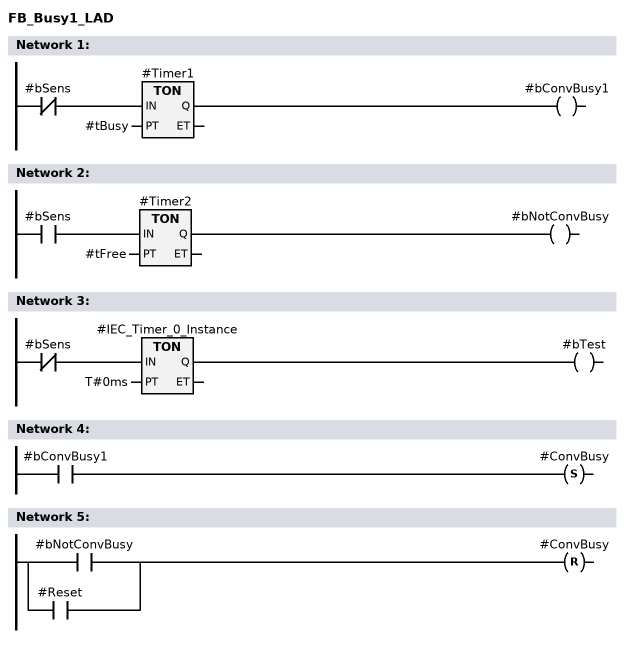
   #Timer1(IN := NOT #bSens, PT := #tBusy);   // TON
   #bConvBusy1 := #Timer1.Q;
END_REGION

REGION Network 2
   #Timer2(IN := #bSens, PT := #tFree);   // TON
   #bNotConvBusy := #Timer2.Q;
END_REGION

REGION Network 3
   #IEC_Timer_0_Instance(IN := NOT #bSens, PT := T#0ms);   // TON
   #bTest := #IEC_Timer_0_Instance.Q;
END_REGION

REGION Network 4
   RUNG wire#powerrail
      Contact( #bConvBusy1 )
      S_Coil( #ConvBusy )
   END_RUNG
   // the same network as SCL:
   IF #bConvBusy1 THEN #ConvBusy := TRUE; END_IF;
END_REGION

REGION Network 5
   RUNG wire#powerrail
      Contact( #bNotConvBusy )
      wire#w1
      R_Coil( #ConvBusy )
   END_RUNG
   RUNG wire#powerrail
      Contact( #Reset )
   END_RUNG wire#w1
   // the same network as SCL:
   IF #bNotConvBusy OR #Reset THEN #ConvBusy := FALSE; END_IF;
END_REGION
END_FUNCTION_BLOCK

FUNCTION_BLOCK "FB_Button"   // FB9, LAD
{ S7_Optimized_Access := 'FALSE' }
VERSION : 0.1
   VAR_INPUT
      bBut : Bool;
      bRS : Bool;
      bJogMode : Bool := false;
      tOnTime : Time := T#3000ms;
   END_VAR
   VAR_OUTPUT
      bOutB : Bool;
   END_VAR
   VAR
      bM : Bool;
      bM1 : Bool;
      bM2 : Bool;
      bM3 : Bool;
      bM4 : Bool;
      bOutBMem : Bool;
      bTemp : Bool;
      IEC_Timer_0_Instance : TON_TIME;
   END_VAR
   VAR_TEMP   // added for the SCL form of the ladder/FBD networks
      _w1 : Bool;
   END_VAR
BEGIN

REGION Network 1
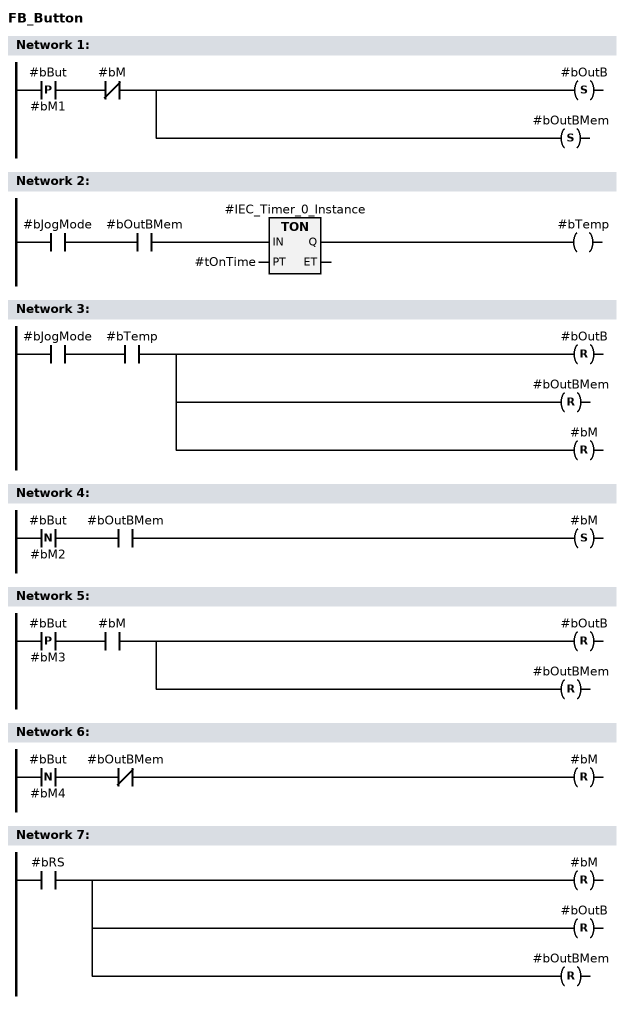
   RUNG wire#powerrail
      P_Contact(operand := #bBut, bit := #bM1)
      I_Contact( #bM )
      wire#w1
      S_Coil( #bOutB )
   END_RUNG
   RUNG wire#w1
      S_Coil( #bOutBMem )
   END_RUNG
   // the same network as SCL:
   #_w1 := #bBut AND NOT #bM1;   // rising edge of #bBut
   #bM1 := #bBut;
   IF #_w1 AND NOT #bM THEN
       #bOutB := TRUE;
       #bOutBMem := TRUE;
   END_IF;
END_REGION

REGION Network 2
   #IEC_Timer_0_Instance(IN := #bJogMode AND #bOutBMem, PT := #tOnTime);   // TON
   #bTemp := #IEC_Timer_0_Instance.Q;
END_REGION

REGION Network 3
   RUNG wire#powerrail
      Contact( #bJogMode )
      Contact( #bTemp )
      wire#w1
      R_Coil( #bOutB )
   END_RUNG
   RUNG wire#w1
      R_Coil( #bOutBMem )
   END_RUNG
   RUNG wire#w1
      R_Coil( #bM )
   END_RUNG
   // the same network as SCL:
   IF #bJogMode AND #bTemp THEN
       #bOutB := FALSE;
       #bOutBMem := FALSE;
       #bM := FALSE;
   END_IF;
END_REGION

REGION Network 4
   RUNG wire#powerrail
      N_Contact(operand := #bBut, bit := #bM2)
      Contact( #bOutBMem )
      S_Coil( #bM )
   END_RUNG
   // the same network as SCL:
   #_w1 := NOT #bBut AND #bM2;   // falling edge of #bBut
   #bM2 := #bBut;
   IF #_w1 AND #bOutBMem THEN #bM := TRUE; END_IF;
END_REGION

REGION Network 5
   RUNG wire#powerrail
      P_Contact(operand := #bBut, bit := #bM3)
      Contact( #bM )
      wire#w1
      R_Coil( #bOutB )
   END_RUNG
   RUNG wire#w1
      R_Coil( #bOutBMem )
   END_RUNG
   // the same network as SCL:
   #_w1 := #bBut AND NOT #bM3;   // rising edge of #bBut
   #bM3 := #bBut;
   IF #_w1 AND #bM THEN
       #bOutB := FALSE;
       #bOutBMem := FALSE;
   END_IF;
END_REGION

REGION Network 6
   RUNG wire#powerrail
      N_Contact(operand := #bBut, bit := #bM4)
      I_Contact( #bOutBMem )
      R_Coil( #bM )
   END_RUNG
   // the same network as SCL:
   #_w1 := NOT #bBut AND #bM4;   // falling edge of #bBut
   #bM4 := #bBut;
   IF #_w1 AND NOT #bOutBMem THEN #bM := FALSE; END_IF;
END_REGION

REGION Network 7
   RUNG wire#powerrail
      Contact( #bRS )
      wire#w1
      R_Coil( #bM )
   END_RUNG
   RUNG wire#w1
      R_Coil( #bOutB )
   END_RUNG
   RUNG wire#w1
      R_Coil( #bOutBMem )
   END_RUNG
   // the same network as SCL:
   IF #bRS THEN
       #bM := FALSE;
       #bOutB := FALSE;
       #bOutBMem := FALSE;
   END_IF;
END_REGION
END_FUNCTION_BLOCK

FUNCTION_BLOCK "FB_Busy2_LAD"   // FB10, LAD
{ S7_Optimized_Access := 'FALSE' }
VERSION : 0.1
// Фильтр для индуктивного датчика
   VAR_INPUT
      bSens : Bool;
      tBusy : Time;
      tFree : Time;
      Reset : Bool;
   END_VAR
   VAR_OUTPUT
      ConvBusy : Bool;
   END_VAR
   VAR
      bConvBusy1 : Bool := false;
      bNotConvBusy : Bool;
      Timer1 : TON_TIME;
      Timer2 : TON_TIME;
   END_VAR
BEGIN

REGION Network 1
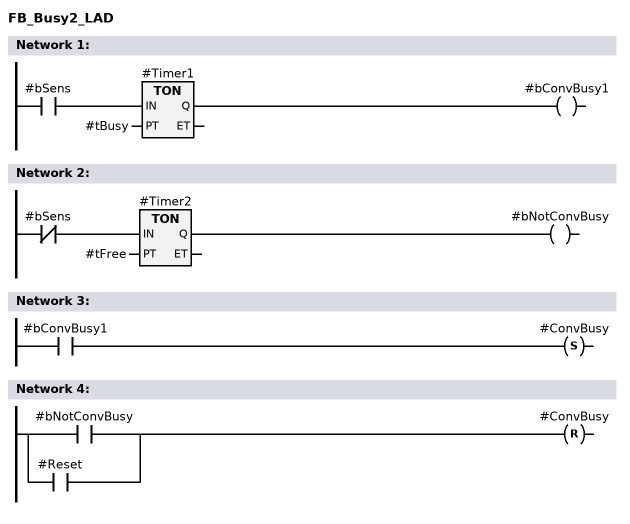
   #Timer1(IN := #bSens, PT := #tBusy);   // TON
   #bConvBusy1 := #Timer1.Q;
END_REGION

REGION Network 2
   #Timer2(IN := NOT #bSens, PT := #tFree);   // TON
   #bNotConvBusy := #Timer2.Q;
END_REGION

REGION Network 3
   RUNG wire#powerrail
      Contact( #bConvBusy1 )
      S_Coil( #ConvBusy )
   END_RUNG
   // the same network as SCL:
   IF #bConvBusy1 THEN #ConvBusy := TRUE; END_IF;
END_REGION

REGION Network 4
   RUNG wire#powerrail
      Contact( #bNotConvBusy )
      wire#w1
      R_Coil( #ConvBusy )
   END_RUNG
   RUNG wire#powerrail
      Contact( #Reset )
   END_RUNG wire#w1
   // the same network as SCL:
   IF #bNotConvBusy OR #Reset THEN #ConvBusy := FALSE; END_IF;
END_REGION
END_FUNCTION_BLOCK

FUNCTION_BLOCK "FB_r_trig"   // FB11, LAD
{ S7_Optimized_Access := 'FALSE' }
VERSION : 0.1
   VAR_INPUT
      CLK : Bool;
   END_VAR
   VAR_OUTPUT
      Q : Bool;
   END_VAR
   VAR
      bR : Bool;
   END_VAR
   VAR_TEMP   // added for the SCL form of the ladder/FBD networks
      _w1 : Bool;
   END_VAR
BEGIN

REGION Network 1
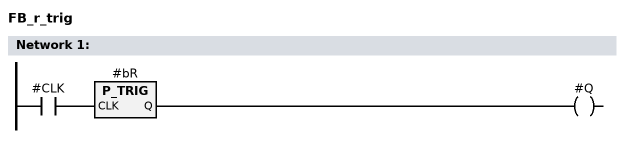
   RUNG wire#powerrail
      Contact( #CLK )
      P_Trig( #bR )
      Coil( #Q )
   END_RUNG
   // the same network as SCL:
   #_w1 := #CLK AND NOT #bR;   // rising edge
   #bR := #CLK;
   #Q := #_w1;
END_REGION
END_FUNCTION_BLOCK

FUNCTION_BLOCK "FB_Move1"   // FB12, LAD
{ S7_Optimized_Access := 'FALSE' }
VERSION : 0.1
   VAR_INPUT
      bConvPlacePos1 : Bool;
      bConvPlacePos2 : Bool;
      tLongMove : Time;
      bEnable1 : Bool;
      bEnable2 : Bool;
      bReset : Bool;
      bStop : Bool;
   END_VAR
   VAR_OUTPUT
      bDrive : Bool;
      bLongMove : Bool;
   END_VAR
   VAR_IN_OUT
      bMove : Bool;
   END_VAR
   VAR
      fbLongMove : TON_TIME;
   END_VAR
BEGIN

REGION Network 1
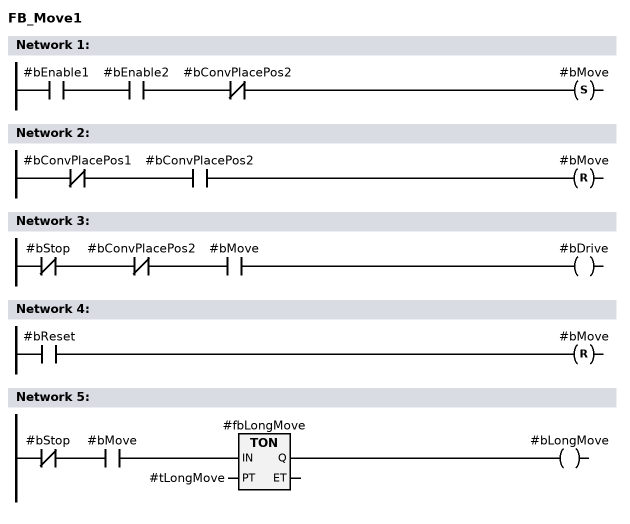
   RUNG wire#powerrail
      Contact( #bEnable1 )
      Contact( #bEnable2 )
      I_Contact( #bConvPlacePos2 )
      S_Coil( #bMove )
   END_RUNG
   // the same network as SCL:
   IF #bEnable1 AND #bEnable2 AND NOT #bConvPlacePos2 THEN #bMove := TRUE; END_IF;
END_REGION

REGION Network 2
   RUNG wire#powerrail
      I_Contact( #bConvPlacePos1 )
      Contact( #bConvPlacePos2 )
      R_Coil( #bMove )
   END_RUNG
   // the same network as SCL:
   IF NOT #bConvPlacePos1 AND #bConvPlacePos2 THEN #bMove := FALSE; END_IF;
END_REGION

REGION Network 3
   RUNG wire#powerrail
      I_Contact( #bStop )
      I_Contact( #bConvPlacePos2 )
      Contact( #bMove )
      Coil( #bDrive )
   END_RUNG
   // the same network as SCL:
   #bDrive := NOT #bStop AND NOT #bConvPlacePos2 AND #bMove;
END_REGION

REGION Network 4
   RUNG wire#powerrail
      Contact( #bReset )
      R_Coil( #bMove )
   END_RUNG
   // the same network as SCL:
   IF #bReset THEN #bMove := FALSE; END_IF;
END_REGION

REGION Network 5
   #fbLongMove(IN := NOT #bStop AND #bMove, PT := #tLongMove);   // TON
   #bLongMove := #fbLongMove.Q;
END_REGION
END_FUNCTION_BLOCK

// folder: Safety

